REGION Network 7: FIXTURES NO DEFINE POSITION
   RUNG wire#powerrail
      Contact( "M_ONE" )
      wire#w1
      I_Contact( "DB4000_FIX_TABLE_POSITIONS".UNIT_01.FIXTURE_1.IN_LOAD_UNLOAD_STATION_1 )
      I_Contact( "DB4000_FIX_TABLE_POSITIONS".UNIT_01.FIXTURE_1.IN_SPARE_STATION_2 )
      I_Contact( "DB4000_FIX_TABLE_POSITIONS".UNIT_01.FIXTURE_1.IN_CLADDING_STATION_3 )
      I_Contact( "DB4000_FIX_TABLE_POSITIONS".UNIT_01.FIXTURE_1.IN_CLEAN_STATION_4 )
      Coil( "DB4000_FIX_TABLE_POSITIONS".UNIT_01.FIXTURE_1.NO_DEFINED_POSITION )
   END_RUNG
   RUNG wire#w1
      I_Contact( "DB4000_FIX_TABLE_POSITIONS".UNIT_01.FIXTURE_2.IN_LOAD_UNLOAD_STATION_1 )
      I_Contact( "DB4000_FIX_TABLE_POSITIONS".UNIT_01.FIXTURE_2.IN_SPARE_STATION_2 )
      I_Contact( "DB4000_FIX_TABLE_POSITIONS".UNIT_01.FIXTURE_2.IN_CLADDING_STATION_3 )
      I_Contact( "DB4000_FIX_TABLE_POSITIONS".UNIT_01.FIXTURE_2.IN_CLEAN_STATION_4 )
      Coil( "DB4000_FIX_TABLE_POSITIONS".UNIT_01.FIXTURE_2.NO_DEFINED_POSITION )
   END_RUNG
   RUNG wire#w1
      I_Contact( "DB4000_FIX_TABLE_POSITIONS".UNIT_01.FIXTURE_3.IN_LOAD_UNLOAD_STATION_1 )
      I_Contact( "DB4000_FIX_TABLE_POSITIONS".UNIT_01.FIXTURE_3.IN_SPARE_STATION_2 )
      I_Contact( "DB4000_FIX_TABLE_POSITIONS".UNIT_01.FIXTURE_3.IN_CLADDING_STATION_3 )
      I_Contact( "DB4000_FIX_TABLE_POSITIONS".UNIT_01.FIXTURE_3.IN_CLEAN_STATION_4 )
      Coil( "DB4000_FIX_TABLE_POSITIONS".UNIT_01.FIXTURE_3.NO_DEFINED_POSITION )
   END_RUNG
   RUNG wire#w1
      I_Contact( "DB4000_FIX_TABLE_POSITIONS".UNIT_01.FIXTURE_4.IN_LOAD_UNLOAD_STATION_1 )
      I_Contact( "DB4000_FIX_TABLE_POSITIONS".UNIT_01.FIXTURE_4.IN_SPARE_STATION_2 )
      I_Contact( "DB4000_FIX_TABLE_POSITIONS".UNIT_01.FIXTURE_4.IN_CLADDING_STATION_3 )
      I_Contact( "DB4000_FIX_TABLE_POSITIONS".UNIT_01.FIXTURE_4.IN_CLEAN_STATION_4 )
      Coil( "DB4000_FIX_TABLE_POSITIONS".UNIT_01.FIXTURE_4.NO_DEFINED_POSITION )
   END_RUNG
   // the same network as SCL:
   "DB4000_FIX_TABLE_POSITIONS".UNIT_01.FIXTURE_1.NO_DEFINED_POSITION := "M_ONE" AND NOT "DB4000_FIX_TABLE_POSITIONS".UNIT_01.FIXTURE_1.IN_LOAD_UNLOAD_STATION_1 AND NOT "DB4000_FIX_TABLE_POSITIONS".UNIT_01.FIXTURE_1.IN_SPARE_STATION_2 AND NOT "DB4000_FIX_TABLE_POSITIONS".UNIT_01.FIXTURE_1.IN_CLADDING_STATION_3 AND NOT "DB4000_FIX_TABLE_POSITIONS".UNIT_01.FIXTURE_1.IN_CLEAN_STATION_4;
   "DB4000_FIX_TABLE_POSITIONS".UNIT_01.FIXTURE_2.NO_DEFINED_POSITION := "M_ONE" AND NOT "DB4000_FIX_TABLE_POSITIONS".UNIT_01.FIXTURE_2.IN_LOAD_UNLOAD_STATION_1 AND NOT "DB4000_FIX_TABLE_POSITIONS".UNIT_01.FIXTURE_2.IN_SPARE_STATION_2 AND NOT "DB4000_FIX_TABLE_POSITIONS".UNIT_01.FIXTURE_2.IN_CLADDING_STATION_3 AND NOT "DB4000_FIX_TABLE_POSITIONS".UNIT_01.FIXTURE_2.IN_CLEAN_STATION_4;
   "DB4000_FIX_TABLE_POSITIONS".UNIT_01.FIXTURE_3.NO_DEFINED_POSITION := "M_ONE" AND NOT "DB4000_FIX_TABLE_POSITIONS".UNIT_01.FIXTURE_3.IN_LOAD_UNLOAD_STATION_1 AND NOT "DB4000_FIX_TABLE_POSITIONS".UNIT_01.FIXTURE_3.IN_SPARE_STATION_2 AND NOT "DB4000_FIX_TABLE_POSITIONS".UNIT_01.FIXTURE_3.IN_CLADDING_STATION_3 AND NOT "DB4000_FIX_TABLE_POSITIONS".UNIT_01.FIXTURE_3.IN_CLEAN_STATION_4;
   "DB4000_FIX_TABLE_POSITIONS".UNIT_01.FIXTURE_4.NO_DEFINED_POSITION := "M_ONE" AND NOT "DB4000_FIX_TABLE_POSITIONS".UNIT_01.FIXTURE_4.IN_LOAD_UNLOAD_STATION_1 AND NOT "DB4000_FIX_TABLE_POSITIONS".UNIT_01.FIXTURE_4.IN_SPARE_STATION_2 AND NOT "DB4000_FIX_TABLE_POSITIONS".UNIT_01.FIXTURE_4.IN_CLADDING_STATION_3 AND NOT "DB4000_FIX_TABLE_POSITIONS".UNIT_01.FIXTURE_4.IN_CLEAN_STATION_4;
END_REGION

REGION Network 8: AXIS E10 HOME POSITION
   RUNG wire#powerrail
      I_Contact( "DB131_CLADDING_AXIS_E10".SAFETY_POSITIONS.AX_POS_0_DEGREES.IN_POSITION )
      I_Contact( "DB131_CLADDING_AXIS_E10".SAFETY_POSITIONS.AX_POS_90_DEGREES.IN_POSITION )
      I_Contact( "DB131_CLADDING_AXIS_E10".SAFETY_POSITIONS.AX_POS_180_DEGREES.IN_POSITION )
      I_Contact( "DB131_CLADDING_AXIS_E10".SAFETY_POSITIONS.AX_POS_270_DEGREES.IN_POSITION )
      Not()
      Coil( "DB4000_FIX_TABLE_POSITIONS".UNIT_01.AXIS_E10_HOME_POS )
   END_RUNG
   // the same network as SCL:
   "DB4000_FIX_TABLE_POSITIONS".UNIT_01.AXIS_E10_HOME_POS := NOT (NOT "DB131_CLADDING_AXIS_E10".SAFETY_POSITIONS.AX_POS_0_DEGREES.IN_POSITION AND NOT "DB131_CLADDING_AXIS_E10".SAFETY_POSITIONS.AX_POS_90_DEGREES.IN_POSITION AND NOT "DB131_CLADDING_AXIS_E10".SAFETY_POSITIONS.AX_POS_180_DEGREES.IN_POSITION AND NOT "DB131_CLADDING_AXIS_E10".SAFETY_POSITIONS.AX_POS_270_DEGREES.IN_POSITION);
END_REGION

REGION Network 9: AXIS E10 NOT IN A DEFINED POSITION
   RUNG wire#powerrail
      I_Contact( "DB131_CLADDING_AXIS_E10".SAFETY_POSITIONS.AX_POS_0_DEGREES.IN_POSITION )
      I_Contact( "DB131_CLADDING_AXIS_E10".SAFETY_POSITIONS.AX_POS_90_DEGREES.IN_POSITION )
      I_Contact( "DB131_CLADDING_AXIS_E10".SAFETY_POSITIONS.AX_POS_180_DEGREES.IN_POSITION )
      I_Contact( "DB131_CLADDING_AXIS_E10".SAFETY_POSITIONS.AX_POS_270_DEGREES.IN_POSITION )
      Coil( "DB4000_FIX_TABLE_POSITIONS".UNIT_01.AXIS_E10_NOT_DEFINED_POS )
   END_RUNG
   // the same network as SCL:
   "DB4000_FIX_TABLE_POSITIONS".UNIT_01.AXIS_E10_NOT_DEFINED_POS := NOT "DB131_CLADDING_AXIS_E10".SAFETY_POSITIONS.AX_POS_0_DEGREES.IN_POSITION AND NOT "DB131_CLADDING_AXIS_E10".SAFETY_POSITIONS.AX_POS_90_DEGREES.IN_POSITION AND NOT "DB131_CLADDING_AXIS_E10".SAFETY_POSITIONS.AX_POS_180_DEGREES.IN_POSITION AND NOT "DB131_CLADDING_AXIS_E10".SAFETY_POSITIONS.AX_POS_270_DEGREES.IN_POSITION;
END_REGION

REGION Network 10: <<<<<<<<<<<<<<<<<<<< UNIT 02 >>>>>>>>>>>>>>>>>>>>
END_REGION

REGION Network 11: AXIS E20 0 DEGREES
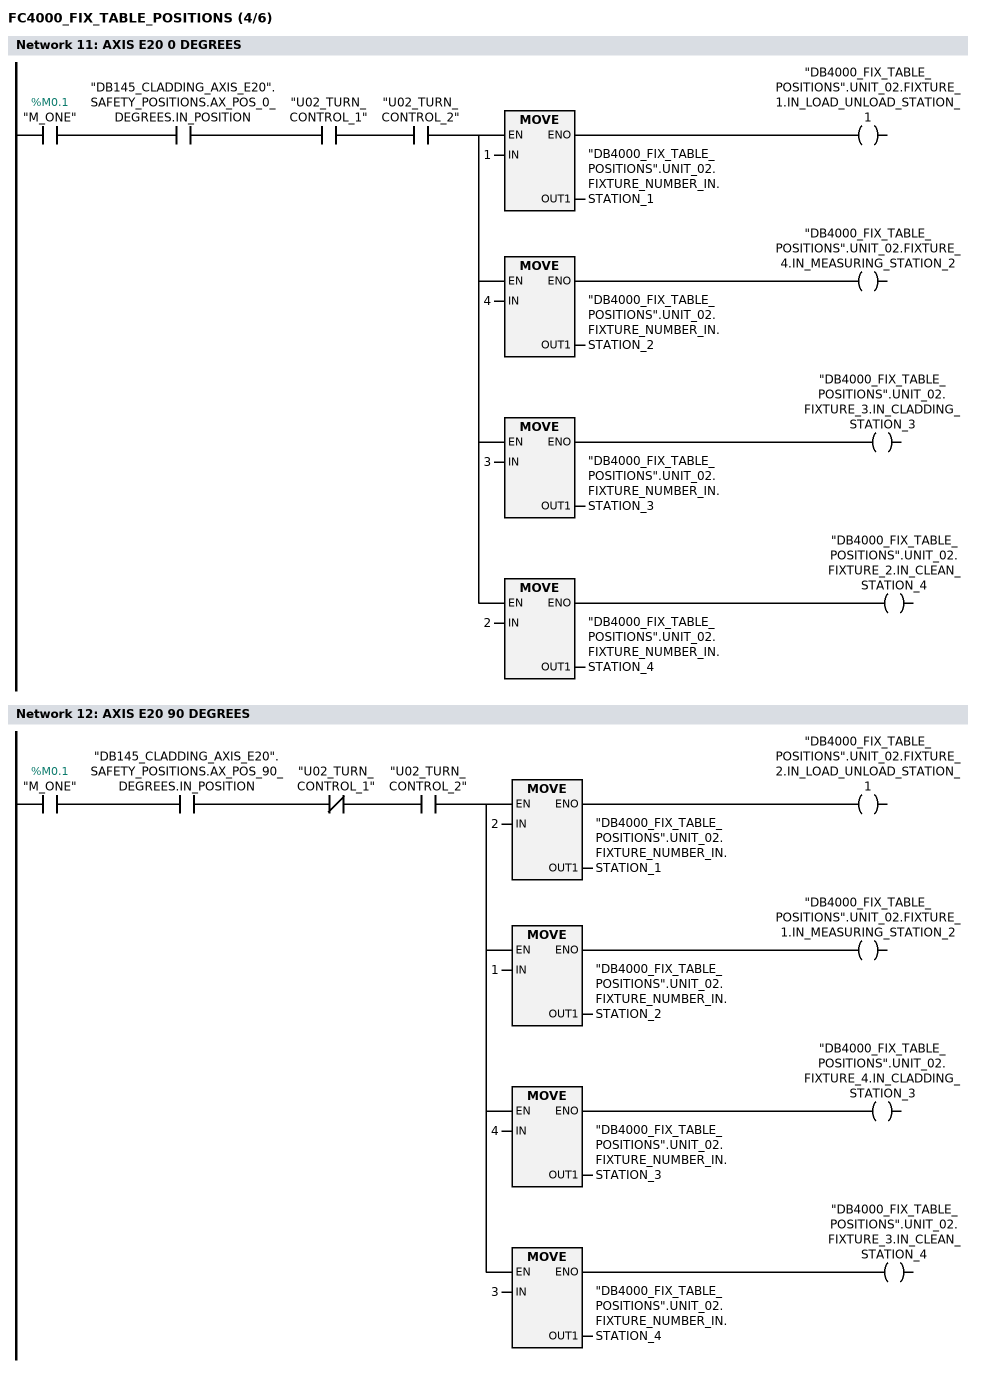
   RUNG wire#powerrail
      Contact( "M_ONE" )
      Contact( "DB145_CLADDING_AXIS_E20".SAFETY_POSITIONS.AX_POS_0_DEGREES.IN_POSITION )
      Contact( "U02_TURN_CONTROL_1" )
      Contact( "U02_TURN_CONTROL_2" )
      wire#w1
      Move(in := 1, out1 => "DB4000_FIX_TABLE_POSITIONS".UNIT_02.FIXTURE_NUMBER_IN.STATION_1)
      Coil( "DB4000_FIX_TABLE_POSITIONS".UNIT_02.FIXTURE_1.IN_LOAD_UNLOAD_STATION_1 )
   END_RUNG
   RUNG wire#w1
      Move(in := 4, out1 => "DB4000_FIX_TABLE_POSITIONS".UNIT_02.FIXTURE_NUMBER_IN.STATION_2)
      Coil( "DB4000_FIX_TABLE_POSITIONS".UNIT_02.FIXTURE_4.IN_MEASURING_STATION_2 )
   END_RUNG
   RUNG wire#w1
      Move(in := 3, out1 => "DB4000_FIX_TABLE_POSITIONS".UNIT_02.FIXTURE_NUMBER_IN.STATION_3)
      Coil( "DB4000_FIX_TABLE_POSITIONS".UNIT_02.FIXTURE_3.IN_CLADDING_STATION_3 )
   END_RUNG
   RUNG wire#w1
      Move(in := 2, out1 => "DB4000_FIX_TABLE_POSITIONS".UNIT_02.FIXTURE_NUMBER_IN.STATION_4)
      Coil( "DB4000_FIX_TABLE_POSITIONS".UNIT_02.FIXTURE_2.IN_CLEAN_STATION_4 )
   END_RUNG
   // the same network as SCL:
   #_w1 := "M_ONE" AND "DB145_CLADDING_AXIS_E20".SAFETY_POSITIONS.AX_POS_0_DEGREES.IN_POSITION AND "U02_TURN_CONTROL_1" AND "U02_TURN_CONTROL_2";
   IF #_w1 THEN "DB4000_FIX_TABLE_POSITIONS".UNIT_02.FIXTURE_NUMBER_IN.STATION_1 := 1; END_IF;
   "DB4000_FIX_TABLE_POSITIONS".UNIT_02.FIXTURE_1.IN_LOAD_UNLOAD_STATION_1 := #_w1;
   IF #_w1 THEN "DB4000_FIX_TABLE_POSITIONS".UNIT_02.FIXTURE_NUMBER_IN.STATION_2 := 4; END_IF;
   "DB4000_FIX_TABLE_POSITIONS".UNIT_02.FIXTURE_4.IN_MEASURING_STATION_2 := #_w1;
   IF #_w1 THEN "DB4000_FIX_TABLE_POSITIONS".UNIT_02.FIXTURE_NUMBER_IN.STATION_3 := 3; END_IF;
   "DB4000_FIX_TABLE_POSITIONS".UNIT_02.FIXTURE_3.IN_CLADDING_STATION_3 := #_w1;
   IF #_w1 THEN "DB4000_FIX_TABLE_POSITIONS".UNIT_02.FIXTURE_NUMBER_IN.STATION_4 := 2; END_IF;
   "DB4000_FIX_TABLE_POSITIONS".UNIT_02.FIXTURE_2.IN_CLEAN_STATION_4 := #_w1;
END_REGION

REGION Network 12: AXIS E20 90 DEGREES
   RUNG wire#powerrail
      Contact( "M_ONE" )
      Contact( "DB145_CLADDING_AXIS_E20".SAFETY_POSITIONS.AX_POS_90_DEGREES.IN_POSITION )
      I_Contact( "U02_TURN_CONTROL_1" )
      Contact( "U02_TURN_CONTROL_2" )
      wire#w1
      Move(in := 2, out1 => "DB4000_FIX_TABLE_POSITIONS".UNIT_02.FIXTURE_NUMBER_IN.STATION_1)
      Coil( "DB4000_FIX_TABLE_POSITIONS".UNIT_02.FIXTURE_2.IN_LOAD_UNLOAD_STATION_1 )
   END_RUNG
   RUNG wire#w1
      Move(in := 1, out1 => "DB4000_FIX_TABLE_POSITIONS".UNIT_02.FIXTURE_NUMBER_IN.STATION_2)
      Coil( "DB4000_FIX_TABLE_POSITIONS".UNIT_02.FIXTURE_1.IN_MEASURING_STATION_2 )
   END_RUNG
   RUNG wire#w1
      Move(in := 4, out1 => "DB4000_FIX_TABLE_POSITIONS".UNIT_02.FIXTURE_NUMBER_IN.STATION_3)
      Coil( "DB4000_FIX_TABLE_POSITIONS".UNIT_02.FIXTURE_4.IN_CLADDING_STATION_3 )
   END_RUNG
   RUNG wire#w1
      Move(in := 3, out1 => "DB4000_FIX_TABLE_POSITIONS".UNIT_02.FIXTURE_NUMBER_IN.STATION_4)
      Coil( "DB4000_FIX_TABLE_POSITIONS".UNIT_02.FIXTURE_3.IN_CLEAN_STATION_4 )
   END_RUNG
   // the same network as SCL:
   #_w1 := "M_ONE" AND "DB145_CLADDING_AXIS_E20".SAFETY_POSITIONS.AX_POS_90_DEGREES.IN_POSITION AND NOT "U02_TURN_CONTROL_1" AND "U02_TURN_CONTROL_2";
   IF #_w1 THEN "DB4000_FIX_TABLE_POSITIONS".UNIT_02.FIXTURE_NUMBER_IN.STATION_1 := 2; END_IF;
   "DB4000_FIX_TABLE_POSITIONS".UNIT_02.FIXTURE_2.IN_LOAD_UNLOAD_STATION_1 := #_w1;
   IF #_w1 THEN "DB4000_FIX_TABLE_POSITIONS".UNIT_02.FIXTURE_NUMBER_IN.STATION_2 := 1; END_IF;
   "DB4000_FIX_TABLE_POSITIONS".UNIT_02.FIXTURE_1.IN_MEASURING_STATION_2 := #_w1;
   IF #_w1 THEN "DB4000_FIX_TABLE_POSITIONS".UNIT_02.FIXTURE_NUMBER_IN.STATION_3 := 4; END_IF;
   "DB4000_FIX_TABLE_POSITIONS".UNIT_02.FIXTURE_4.IN_CLADDING_STATION_3 := #_w1;
   IF #_w1 THEN "DB4000_FIX_TABLE_POSITIONS".UNIT_02.FIXTURE_NUMBER_IN.STATION_4 := 3; END_IF;
   "DB4000_FIX_TABLE_POSITIONS".UNIT_02.FIXTURE_3.IN_CLEAN_STATION_4 := #_w1;
END_REGION

REGION Network 13: AXIS E20 180 DEGREES
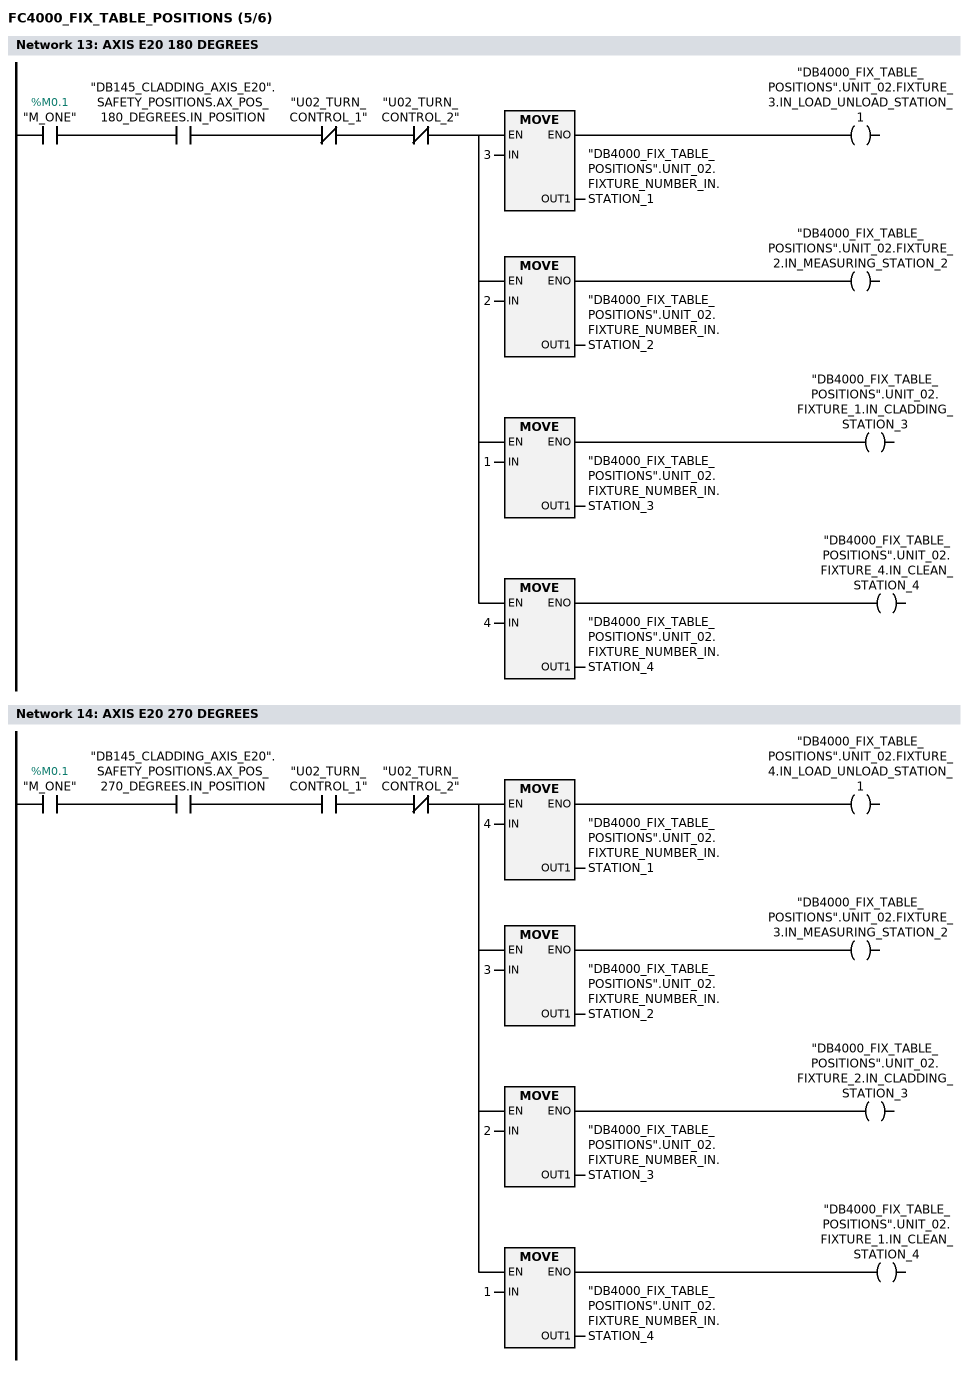
   RUNG wire#powerrail
      Contact( "M_ONE" )
      Contact( "DB145_CLADDING_AXIS_E20".SAFETY_POSITIONS.AX_POS_180_DEGREES.IN_POSITION )
      I_Contact( "U02_TURN_CONTROL_1" )
      I_Contact( "U02_TURN_CONTROL_2" )
      wire#w1
      Move(in := 3, out1 => "DB4000_FIX_TABLE_POSITIONS".UNIT_02.FIXTURE_NUMBER_IN.STATION_1)
      Coil( "DB4000_FIX_TABLE_POSITIONS".UNIT_02.FIXTURE_3.IN_LOAD_UNLOAD_STATION_1 )
   END_RUNG
   RUNG wire#w1
      Move(in := 2, out1 => "DB4000_FIX_TABLE_POSITIONS".UNIT_02.FIXTURE_NUMBER_IN.STATION_2)
      Coil( "DB4000_FIX_TABLE_POSITIONS".UNIT_02.FIXTURE_2.IN_MEASURING_STATION_2 )
   END_RUNG
   RUNG wire#w1
      Move(in := 1, out1 => "DB4000_FIX_TABLE_POSITIONS".UNIT_02.FIXTURE_NUMBER_IN.STATION_3)
      Coil( "DB4000_FIX_TABLE_POSITIONS".UNIT_02.FIXTURE_1.IN_CLADDING_STATION_3 )
   END_RUNG
   RUNG wire#w1
      Move(in := 4, out1 => "DB4000_FIX_TABLE_POSITIONS".UNIT_02.FIXTURE_NUMBER_IN.STATION_4)
      Coil( "DB4000_FIX_TABLE_POSITIONS".UNIT_02.FIXTURE_4.IN_CLEAN_STATION_4 )
   END_RUNG
   // the same network as SCL:
   #_w1 := "M_ONE" AND "DB145_CLADDING_AXIS_E20".SAFETY_POSITIONS.AX_POS_180_DEGREES.IN_POSITION AND NOT "U02_TURN_CONTROL_1" AND NOT "U02_TURN_CONTROL_2";
   IF #_w1 THEN "DB4000_FIX_TABLE_POSITIONS".UNIT_02.FIXTURE_NUMBER_IN.STATION_1 := 3; END_IF;
   "DB4000_FIX_TABLE_POSITIONS".UNIT_02.FIXTURE_3.IN_LOAD_UNLOAD_STATION_1 := #_w1;
   IF #_w1 THEN "DB4000_FIX_TABLE_POSITIONS".UNIT_02.FIXTURE_NUMBER_IN.STATION_2 := 2; END_IF;
   "DB4000_FIX_TABLE_POSITIONS".UNIT_02.FIXTURE_2.IN_MEASURING_STATION_2 := #_w1;
   IF #_w1 THEN "DB4000_FIX_TABLE_POSITIONS".UNIT_02.FIXTURE_NUMBER_IN.STATION_3 := 1; END_IF;
   "DB4000_FIX_TABLE_POSITIONS".UNIT_02.FIXTURE_1.IN_CLADDING_STATION_3 := #_w1;
   IF #_w1 THEN "DB4000_FIX_TABLE_POSITIONS".UNIT_02.FIXTURE_NUMBER_IN.STATION_4 := 4; END_IF;
   "DB4000_FIX_TABLE_POSITIONS".UNIT_02.FIXTURE_4.IN_CLEAN_STATION_4 := #_w1;
END_REGION

REGION Network 14: AXIS E20 270 DEGREES
   RUNG wire#powerrail
      Contact( "M_ONE" )
      Contact( "DB145_CLADDING_AXIS_E20".SAFETY_POSITIONS.AX_POS_270_DEGREES.IN_POSITION )
      Contact( "U02_TURN_CONTROL_1" )
      I_Contact( "U02_TURN_CONTROL_2" )
      wire#w1
      Move(in := 4, out1 => "DB4000_FIX_TABLE_POSITIONS".UNIT_02.FIXTURE_NUMBER_IN.STATION_1)
      Coil( "DB4000_FIX_TABLE_POSITIONS".UNIT_02.FIXTURE_4.IN_LOAD_UNLOAD_STATION_1 )
   END_RUNG
   RUNG wire#w1
      Move(in := 3, out1 => "DB4000_FIX_TABLE_POSITIONS".UNIT_02.FIXTURE_NUMBER_IN.STATION_2)
      Coil( "DB4000_FIX_TABLE_POSITIONS".UNIT_02.FIXTURE_3.IN_MEASURING_STATION_2 )
   END_RUNG
   RUNG wire#w1
      Move(in := 2, out1 => "DB4000_FIX_TABLE_POSITIONS".UNIT_02.FIXTURE_NUMBER_IN.STATION_3)
      Coil( "DB4000_FIX_TABLE_POSITIONS".UNIT_02.FIXTURE_2.IN_CLADDING_STATION_3 )
   END_RUNG
   RUNG wire#w1
      Move(in := 1, out1 => "DB4000_FIX_TABLE_POSITIONS".UNIT_02.FIXTURE_NUMBER_IN.STATION_4)
      Coil( "DB4000_FIX_TABLE_POSITIONS".UNIT_02.FIXTURE_1.IN_CLEAN_STATION_4 )
   END_RUNG
   // the same network as SCL:
   #_w1 := "M_ONE" AND "DB145_CLADDING_AXIS_E20".SAFETY_POSITIONS.AX_POS_270_DEGREES.IN_POSITION AND "U02_TURN_CONTROL_1" AND NOT "U02_TURN_CONTROL_2";
   IF #_w1 THEN "DB4000_FIX_TABLE_POSITIONS".UNIT_02.FIXTURE_NUMBER_IN.STATION_1 := 4; END_IF;
   "DB4000_FIX_TABLE_POSITIONS".UNIT_02.FIXTURE_4.IN_LOAD_UNLOAD_STATION_1 := #_w1;
   IF #_w1 THEN "DB4000_FIX_TABLE_POSITIONS".UNIT_02.FIXTURE_NUMBER_IN.STATION_2 := 3; END_IF;
   "DB4000_FIX_TABLE_POSITIONS".UNIT_02.FIXTURE_3.IN_MEASURING_STATION_2 := #_w1;
   IF #_w1 THEN "DB4000_FIX_TABLE_POSITIONS".UNIT_02.FIXTURE_NUMBER_IN.STATION_3 := 2; END_IF;
   "DB4000_FIX_TABLE_POSITIONS".UNIT_02.FIXTURE_2.IN_CLADDING_STATION_3 := #_w1;
   IF #_w1 THEN "DB4000_FIX_TABLE_POSITIONS".UNIT_02.FIXTURE_NUMBER_IN.STATION_4 := 1; END_IF;
   "DB4000_FIX_TABLE_POSITIONS".UNIT_02.FIXTURE_1.IN_CLEAN_STATION_4 := #_w1;
END_REGION

REGION Network 15: E20 AXIS POSITION REACH
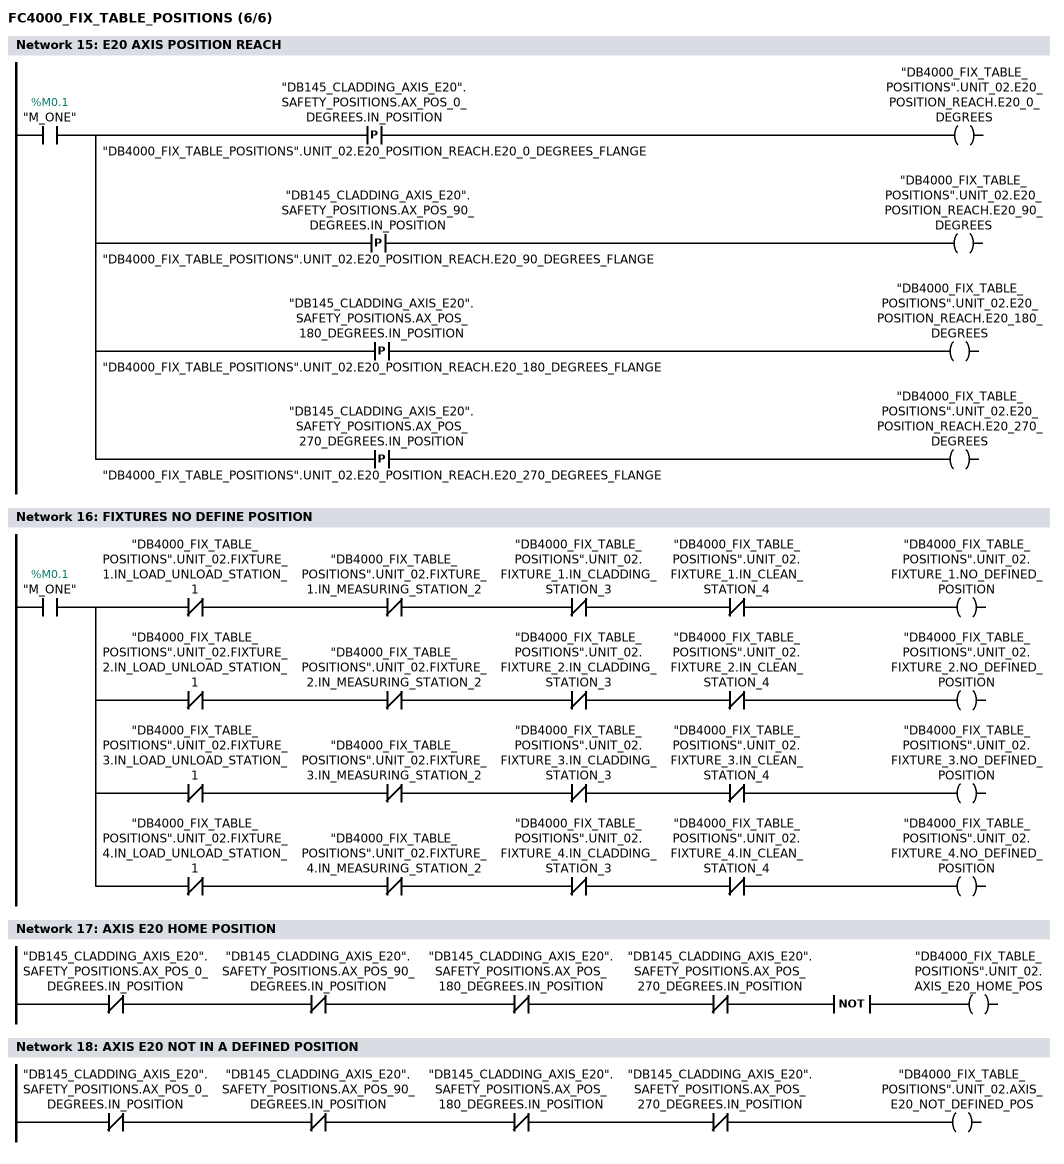
   RUNG wire#powerrail
      Contact( "M_ONE" )
      wire#w1
      P_Contact(operand := "DB145_CLADDING_AXIS_E20".SAFETY_POSITIONS.AX_POS_0_DEGREES.IN_POSITION, bit := "DB4000_FIX_TABLE_POSITIONS".UNIT_02.E20_POSITION_REACH.E20_0_DEGREES_FLANGE)
      Coil( "DB4000_FIX_TABLE_POSITIONS".UNIT_02.E20_POSITION_REACH.E20_0_DEGREES )
   END_RUNG
   RUNG wire#w1
      P_Contact(operand := "DB145_CLADDING_AXIS_E20".SAFETY_POSITIONS.AX_POS_90_DEGREES.IN_POSITION, bit := "DB4000_FIX_TABLE_POSITIONS".UNIT_02.E20_POSITION_REACH.E20_90_DEGREES_FLANGE)
      Coil( "DB4000_FIX_TABLE_POSITIONS".UNIT_02.E20_POSITION_REACH.E20_90_DEGREES )
   END_RUNG
   RUNG wire#w1
      P_Contact(operand := "DB145_CLADDING_AXIS_E20".SAFETY_POSITIONS.AX_POS_180_DEGREES.IN_POSITION, bit := "DB4000_FIX_TABLE_POSITIONS".UNIT_02.E20_POSITION_REACH.E20_180_DEGREES_FLANGE)
      Coil( "DB4000_FIX_TABLE_POSITIONS".UNIT_02.E20_POSITION_REACH.E20_180_DEGREES )
   END_RUNG
   RUNG wire#w1
      P_Contact(operand := "DB145_CLADDING_AXIS_E20".SAFETY_POSITIONS.AX_POS_270_DEGREES.IN_POSITION, bit := "DB4000_FIX_TABLE_POSITIONS".UNIT_02.E20_POSITION_REACH.E20_270_DEGREES_FLANGE)
      Coil( "DB4000_FIX_TABLE_POSITIONS".UNIT_02.E20_POSITION_REACH.E20_270_DEGREES )
   END_RUNG
   // the same network as SCL:
   #_w1 := "M_ONE" AND "DB145_CLADDING_AXIS_E20".SAFETY_POSITIONS.AX_POS_0_DEGREES.IN_POSITION AND NOT "DB4000_FIX_TABLE_POSITIONS".UNIT_02.E20_POSITION_REACH.E20_0_DEGREES_FLANGE;   // rising edge of "DB145_CLADDING_AXIS_E20".SAFETY_POSITIONS.AX_POS_0_DEGREES.IN_POSITION
   "DB4000_FIX_TABLE_POSITIONS".UNIT_02.E20_POSITION_REACH.E20_0_DEGREES_FLANGE := "DB145_CLADDING_AXIS_E20".SAFETY_POSITIONS.AX_POS_0_DEGREES.IN_POSITION;
   "DB4000_FIX_TABLE_POSITIONS".UNIT_02.E20_POSITION_REACH.E20_0_DEGREES := #_w1;
   #_w2 := "M_ONE" AND "DB145_CLADDING_AXIS_E20".SAFETY_POSITIONS.AX_POS_90_DEGREES.IN_POSITION AND NOT "DB4000_FIX_TABLE_POSITIONS".UNIT_02.E20_POSITION_REACH.E20_90_DEGREES_FLANGE;   // rising edge of "DB145_CLADDING_AXIS_E20".SAFETY_POSITIONS.AX_POS_90_DEGREES.IN_POSITION
   "DB4000_FIX_TABLE_POSITIONS".UNIT_02.E20_POSITION_REACH.E20_90_DEGREES_FLANGE := "DB145_CLADDING_AXIS_E20".SAFETY_POSITIONS.AX_POS_90_DEGREES.IN_POSITION;
   "DB4000_FIX_TABLE_POSITIONS".UNIT_02.E20_POSITION_REACH.E20_90_DEGREES := #_w2;
   #_w3 := "M_ONE" AND "DB145_CLADDING_AXIS_E20".SAFETY_POSITIONS.AX_POS_180_DEGREES.IN_POSITION AND NOT "DB4000_FIX_TABLE_POSITIONS".UNIT_02.E20_POSITION_REACH.E20_180_DEGREES_FLANGE;   // rising edge of "DB145_CLADDING_AXIS_E20".SAFETY_POSITIONS.AX_POS_180_DEGREES.IN_POSITION
   "DB4000_FIX_TABLE_POSITIONS".UNIT_02.E20_POSITION_REACH.E20_180_DEGREES_FLANGE := "DB145_CLADDING_AXIS_E20".SAFETY_POSITIONS.AX_POS_180_DEGREES.IN_POSITION;
   "DB4000_FIX_TABLE_POSITIONS".UNIT_02.E20_POSITION_REACH.E20_180_DEGREES := #_w3;
   #_w4 := "M_ONE" AND "DB145_CLADDING_AXIS_E20".SAFETY_POSITIONS.AX_POS_270_DEGREES.IN_POSITION AND NOT "DB4000_FIX_TABLE_POSITIONS".UNIT_02.E20_POSITION_REACH.E20_270_DEGREES_FLANGE;   // rising edge of "DB145_CLADDING_AXIS_E20".SAFETY_POSITIONS.AX_POS_270_DEGREES.IN_POSITION
   "DB4000_FIX_TABLE_POSITIONS".UNIT_02.E20_POSITION_REACH.E20_270_DEGREES_FLANGE := "DB145_CLADDING_AXIS_E20".SAFETY_POSITIONS.AX_POS_270_DEGREES.IN_POSITION;
   "DB4000_FIX_TABLE_POSITIONS".UNIT_02.E20_POSITION_REACH.E20_270_DEGREES := #_w4;
END_REGION

REGION Network 16: FIXTURES NO DEFINE POSITION
   RUNG wire#powerrail
      Contact( "M_ONE" )
      wire#w1
      I_Contact( "DB4000_FIX_TABLE_POSITIONS".UNIT_02.FIXTURE_1.IN_LOAD_UNLOAD_STATION_1 )
      I_Contact( "DB4000_FIX_TABLE_POSITIONS".UNIT_02.FIXTURE_1.IN_MEASURING_STATION_2 )
      I_Contact( "DB4000_FIX_TABLE_POSITIONS".UNIT_02.FIXTURE_1.IN_CLADDING_STATION_3 )
      I_Contact( "DB4000_FIX_TABLE_POSITIONS".UNIT_02.FIXTURE_1.IN_CLEAN_STATION_4 )
      Coil( "DB4000_FIX_TABLE_POSITIONS".UNIT_02.FIXTURE_1.NO_DEFINED_POSITION )
   END_RUNG
   RUNG wire#w1
      I_Contact( "DB4000_FIX_TABLE_POSITIONS".UNIT_02.FIXTURE_2.IN_LOAD_UNLOAD_STATION_1 )
      I_Contact( "DB4000_FIX_TABLE_POSITIONS".UNIT_02.FIXTURE_2.IN_MEASURING_STATION_2 )
      I_Contact( "DB4000_FIX_TABLE_POSITIONS".UNIT_02.FIXTURE_2.IN_CLADDING_STATION_3 )
      I_Contact( "DB4000_FIX_TABLE_POSITIONS".UNIT_02.FIXTURE_2.IN_CLEAN_STATION_4 )
      Coil( "DB4000_FIX_TABLE_POSITIONS".UNIT_02.FIXTURE_2.NO_DEFINED_POSITION )
   END_RUNG
   RUNG wire#w1
      I_Contact( "DB4000_FIX_TABLE_POSITIONS".UNIT_02.FIXTURE_3.IN_LOAD_UNLOAD_STATION_1 )
      I_Contact( "DB4000_FIX_TABLE_POSITIONS".UNIT_02.FIXTURE_3.IN_MEASURING_STATION_2 )
      I_Contact( "DB4000_FIX_TABLE_POSITIONS".UNIT_02.FIXTURE_3.IN_CLADDING_STATION_3 )
      I_Contact( "DB4000_FIX_TABLE_POSITIONS".UNIT_02.FIXTURE_3.IN_CLEAN_STATION_4 )
      Coil( "DB4000_FIX_TABLE_POSITIONS".UNIT_02.FIXTURE_3.NO_DEFINED_POSITION )
   END_RUNG
   RUNG wire#w1
      I_Contact( "DB4000_FIX_TABLE_POSITIONS".UNIT_02.FIXTURE_4.IN_LOAD_UNLOAD_STATION_1 )
      I_Contact( "DB4000_FIX_TABLE_POSITIONS".UNIT_02.FIXTURE_4.IN_MEASURING_STATION_2 )
      I_Contact( "DB4000_FIX_TABLE_POSITIONS".UNIT_02.FIXTURE_4.IN_CLADDING_STATION_3 )
      I_Contact( "DB4000_FIX_TABLE_POSITIONS".UNIT_02.FIXTURE_4.IN_CLEAN_STATION_4 )
      Coil( "DB4000_FIX_TABLE_POSITIONS".UNIT_02.FIXTURE_4.NO_DEFINED_POSITION )
   END_RUNG
   // the same network as SCL:
   "DB4000_FIX_TABLE_POSITIONS".UNIT_02.FIXTURE_1.NO_DEFINED_POSITION := "M_ONE" AND NOT "DB4000_FIX_TABLE_POSITIONS".UNIT_02.FIXTURE_1.IN_LOAD_UNLOAD_STATION_1 AND NOT "DB4000_FIX_TABLE_POSITIONS".UNIT_02.FIXTURE_1.IN_MEASURING_STATION_2 AND NOT "DB4000_FIX_TABLE_POSITIONS".UNIT_02.FIXTURE_1.IN_CLADDING_STATION_3 AND NOT "DB4000_FIX_TABLE_POSITIONS".UNIT_02.FIXTURE_1.IN_CLEAN_STATION_4;
   "DB4000_FIX_TABLE_POSITIONS".UNIT_02.FIXTURE_2.NO_DEFINED_POSITION := "M_ONE" AND NOT "DB4000_FIX_TABLE_POSITIONS".UNIT_02.FIXTURE_2.IN_LOAD_UNLOAD_STATION_1 AND NOT "DB4000_FIX_TABLE_POSITIONS".UNIT_02.FIXTURE_2.IN_MEASURING_STATION_2 AND NOT "DB4000_FIX_TABLE_POSITIONS".UNIT_02.FIXTURE_2.IN_CLADDING_STATION_3 AND NOT "DB4000_FIX_TABLE_POSITIONS".UNIT_02.FIXTURE_2.IN_CLEAN_STATION_4;
   "DB4000_FIX_TABLE_POSITIONS".UNIT_02.FIXTURE_3.NO_DEFINED_POSITION := "M_ONE" AND NOT "DB4000_FIX_TABLE_POSITIONS".UNIT_02.FIXTURE_3.IN_LOAD_UNLOAD_STATION_1 AND NOT "DB4000_FIX_TABLE_POSITIONS".UNIT_02.FIXTURE_3.IN_MEASURING_STATION_2 AND NOT "DB4000_FIX_TABLE_POSITIONS".UNIT_02.FIXTURE_3.IN_CLADDING_STATION_3 AND NOT "DB4000_FIX_TABLE_POSITIONS".UNIT_02.FIXTURE_3.IN_CLEAN_STATION_4;
   "DB4000_FIX_TABLE_POSITIONS".UNIT_02.FIXTURE_4.NO_DEFINED_POSITION := "M_ONE" AND NOT "DB4000_FIX_TABLE_POSITIONS".UNIT_02.FIXTURE_4.IN_LOAD_UNLOAD_STATION_1 AND NOT "DB4000_FIX_TABLE_POSITIONS".UNIT_02.FIXTURE_4.IN_MEASURING_STATION_2 AND NOT "DB4000_FIX_TABLE_POSITIONS".UNIT_02.FIXTURE_4.IN_CLADDING_STATION_3 AND NOT "DB4000_FIX_TABLE_POSITIONS".UNIT_02.FIXTURE_4.IN_CLEAN_STATION_4;
END_REGION

REGION Network 17: AXIS E20 HOME POSITION
   RUNG wire#powerrail
      I_Contact( "DB145_CLADDING_AXIS_E20".SAFETY_POSITIONS.AX_POS_0_DEGREES.IN_POSITION )
      I_Contact( "DB145_CLADDING_AXIS_E20".SAFETY_POSITIONS.AX_POS_90_DEGREES.IN_POSITION )
      I_Contact( "DB145_CLADDING_AXIS_E20".SAFETY_POSITIONS.AX_POS_180_DEGREES.IN_POSITION )
      I_Contact( "DB145_CLADDING_AXIS_E20".SAFETY_POSITIONS.AX_POS_270_DEGREES.IN_POSITION )
      Not()
      Coil( "DB4000_FIX_TABLE_POSITIONS".UNIT_02.AXIS_E20_HOME_POS )
   END_RUNG
   // the same network as SCL:
   "DB4000_FIX_TABLE_POSITIONS".UNIT_02.AXIS_E20_HOME_POS := NOT (NOT "DB145_CLADDING_AXIS_E20".SAFETY_POSITIONS.AX_POS_0_DEGREES.IN_POSITION AND NOT "DB145_CLADDING_AXIS_E20".SAFETY_POSITIONS.AX_POS_90_DEGREES.IN_POSITION AND NOT "DB145_CLADDING_AXIS_E20".SAFETY_POSITIONS.AX_POS_180_DEGREES.IN_POSITION AND NOT "DB145_CLADDING_AXIS_E20".SAFETY_POSITIONS.AX_POS_270_DEGREES.IN_POSITION);
END_REGION

REGION Network 18: AXIS E20 NOT IN A DEFINED POSITION
   RUNG wire#powerrail
      I_Contact( "DB145_CLADDING_AXIS_E20".SAFETY_POSITIONS.AX_POS_0_DEGREES.IN_POSITION )
      I_Contact( "DB145_CLADDING_AXIS_E20".SAFETY_POSITIONS.AX_POS_90_DEGREES.IN_POSITION )
      I_Contact( "DB145_CLADDING_AXIS_E20".SAFETY_POSITIONS.AX_POS_180_DEGREES.IN_POSITION )
      I_Contact( "DB145_CLADDING_AXIS_E20".SAFETY_POSITIONS.AX_POS_270_DEGREES.IN_POSITION )
      Coil( "DB4000_FIX_TABLE_POSITIONS".UNIT_02.AXIS_E20_NOT_DEFINED_POS )
   END_RUNG
   // the same network as SCL:
   "DB4000_FIX_TABLE_POSITIONS".UNIT_02.AXIS_E20_NOT_DEFINED_POS := NOT "DB145_CLADDING_AXIS_E20".SAFETY_POSITIONS.AX_POS_0_DEGREES.IN_POSITION AND NOT "DB145_CLADDING_AXIS_E20".SAFETY_POSITIONS.AX_POS_90_DEGREES.IN_POSITION AND NOT "DB145_CLADDING_AXIS_E20".SAFETY_POSITIONS.AX_POS_180_DEGREES.IN_POSITION AND NOT "DB145_CLADDING_AXIS_E20".SAFETY_POSITIONS.AX_POS_270_DEGREES.IN_POSITION;
END_REGION
END_FUNCTION

FUNCTION "FC4001_FIXTURES_CALIBRATION" : Void   // FC4001, LAD
{ S7_Optimized_Access := 'TRUE' }
VERSION : 0.1
// stored: AutoNumber false, IsIECCheckEnabled false, SetENOAutomatically false, UDAEnableTagReadback false
BEGIN

REGION Network 1: FIXTURE 1 STATION 2 CALIBRATION DONE MEMORY
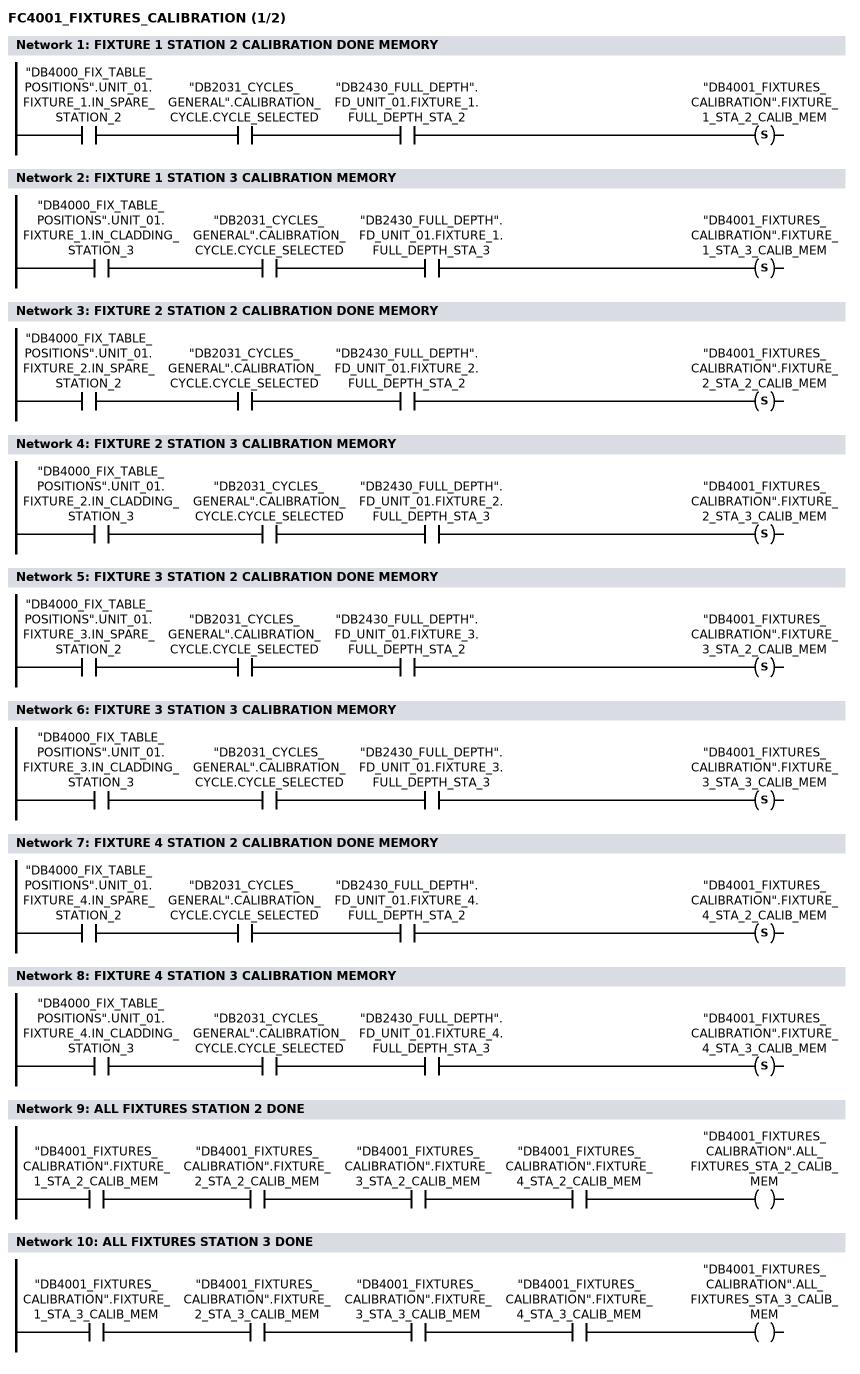
   RUNG wire#powerrail
      Contact( "DB4000_FIX_TABLE_POSITIONS".UNIT_01.FIXTURE_1.IN_SPARE_STATION_2 )
      Contact( "DB2031_CYCLES_GENERAL".CALIBRATION_CYCLE.CYCLE_SELECTED )
      Contact( "DB2430_FULL_DEPTH".FD_UNIT_01.FIXTURE_1.FULL_DEPTH_STA_2 )
      S_Coil( "DB4001_FIXTURES_CALIBRATION".FIXTURE_1_STA_2_CALIB_MEM )
   END_RUNG
   // the same network as SCL:
   IF "DB4000_FIX_TABLE_POSITIONS".UNIT_01.FIXTURE_1.IN_SPARE_STATION_2 AND "DB2031_CYCLES_GENERAL".CALIBRATION_CYCLE.CYCLE_SELECTED AND "DB2430_FULL_DEPTH".FD_UNIT_01.FIXTURE_1.FULL_DEPTH_STA_2 THEN
       "DB4001_FIXTURES_CALIBRATION".FIXTURE_1_STA_2_CALIB_MEM := TRUE;
   END_IF;
END_REGION

REGION Network 2: FIXTURE 1 STATION 3 CALIBRATION MEMORY
   RUNG wire#powerrail
      Contact( "DB4000_FIX_TABLE_POSITIONS".UNIT_01.FIXTURE_1.IN_CLADDING_STATION_3 )
      Contact( "DB2031_CYCLES_GENERAL".CALIBRATION_CYCLE.CYCLE_SELECTED )
      Contact( "DB2430_FULL_DEPTH".FD_UNIT_01.FIXTURE_1.FULL_DEPTH_STA_3 )
      S_Coil( "DB4001_FIXTURES_CALIBRATION".FIXTURE_1_STA_3_CALIB_MEM )
   END_RUNG
   // the same network as SCL:
   IF "DB4000_FIX_TABLE_POSITIONS".UNIT_01.FIXTURE_1.IN_CLADDING_STATION_3 AND "DB2031_CYCLES_GENERAL".CALIBRATION_CYCLE.CYCLE_SELECTED AND "DB2430_FULL_DEPTH".FD_UNIT_01.FIXTURE_1.FULL_DEPTH_STA_3 THEN
       "DB4001_FIXTURES_CALIBRATION".FIXTURE_1_STA_3_CALIB_MEM := TRUE;
   END_IF;
END_REGION

REGION Network 3: FIXTURE 2 STATION 2 CALIBRATION DONE MEMORY
   RUNG wire#powerrail
      Contact( "DB4000_FIX_TABLE_POSITIONS".UNIT_01.FIXTURE_2.IN_SPARE_STATION_2 )
      Contact( "DB2031_CYCLES_GENERAL".CALIBRATION_CYCLE.CYCLE_SELECTED )
      Contact( "DB2430_FULL_DEPTH".FD_UNIT_01.FIXTURE_2.FULL_DEPTH_STA_2 )
      S_Coil( "DB4001_FIXTURES_CALIBRATION".FIXTURE_2_STA_2_CALIB_MEM )
   END_RUNG
   // the same network as SCL:
   IF "DB4000_FIX_TABLE_POSITIONS".UNIT_01.FIXTURE_2.IN_SPARE_STATION_2 AND "DB2031_CYCLES_GENERAL".CALIBRATION_CYCLE.CYCLE_SELECTED AND "DB2430_FULL_DEPTH".FD_UNIT_01.FIXTURE_2.FULL_DEPTH_STA_2 THEN
       "DB4001_FIXTURES_CALIBRATION".FIXTURE_2_STA_2_CALIB_MEM := TRUE;
   END_IF;
END_REGION

REGION Network 4: FIXTURE 2 STATION 3 CALIBRATION MEMORY
   RUNG wire#powerrail
      Contact( "DB4000_FIX_TABLE_POSITIONS".UNIT_01.FIXTURE_2.IN_CLADDING_STATION_3 )
      Contact( "DB2031_CYCLES_GENERAL".CALIBRATION_CYCLE.CYCLE_SELECTED )
      Contact( "DB2430_FULL_DEPTH".FD_UNIT_01.FIXTURE_2.FULL_DEPTH_STA_3 )
      S_Coil( "DB4001_FIXTURES_CALIBRATION".FIXTURE_2_STA_3_CALIB_MEM )
   END_RUNG
   // the same network as SCL:
   IF "DB4000_FIX_TABLE_POSITIONS".UNIT_01.FIXTURE_2.IN_CLADDING_STATION_3 AND "DB2031_CYCLES_GENERAL".CALIBRATION_CYCLE.CYCLE_SELECTED AND "DB2430_FULL_DEPTH".FD_UNIT_01.FIXTURE_2.FULL_DEPTH_STA_3 THEN
       "DB4001_FIXTURES_CALIBRATION".FIXTURE_2_STA_3_CALIB_MEM := TRUE;
   END_IF;
END_REGION

REGION Network 5: FIXTURE 3 STATION 2 CALIBRATION DONE MEMORY
   RUNG wire#powerrail
      Contact( "DB4000_FIX_TABLE_POSITIONS".UNIT_01.FIXTURE_3.IN_SPARE_STATION_2 )
      Contact( "DB2031_CYCLES_GENERAL".CALIBRATION_CYCLE.CYCLE_SELECTED )
      Contact( "DB2430_FULL_DEPTH".FD_UNIT_01.FIXTURE_3.FULL_DEPTH_STA_2 )
      S_Coil( "DB4001_FIXTURES_CALIBRATION".FIXTURE_3_STA_2_CALIB_MEM )
   END_RUNG
   // the same network as SCL:
   IF "DB4000_FIX_TABLE_POSITIONS".UNIT_01.FIXTURE_3.IN_SPARE_STATION_2 AND "DB2031_CYCLES_GENERAL".CALIBRATION_CYCLE.CYCLE_SELECTED AND "DB2430_FULL_DEPTH".FD_UNIT_01.FIXTURE_3.FULL_DEPTH_STA_2 THEN
       "DB4001_FIXTURES_CALIBRATION".FIXTURE_3_STA_2_CALIB_MEM := TRUE;
   END_IF;
END_REGION

REGION Network 6: FIXTURE 3 STATION 3 CALIBRATION MEMORY
   RUNG wire#powerrail
      Contact( "DB4000_FIX_TABLE_POSITIONS".UNIT_01.FIXTURE_3.IN_CLADDING_STATION_3 )
      Contact( "DB2031_CYCLES_GENERAL".CALIBRATION_CYCLE.CYCLE_SELECTED )
      Contact( "DB2430_FULL_DEPTH".FD_UNIT_01.FIXTURE_3.FULL_DEPTH_STA_3 )
      S_Coil( "DB4001_FIXTURES_CALIBRATION".FIXTURE_3_STA_3_CALIB_MEM )
   END_RUNG
   // the same network as SCL:
   IF "DB4000_FIX_TABLE_POSITIONS".UNIT_01.FIXTURE_3.IN_CLADDING_STATION_3 AND "DB2031_CYCLES_GENERAL".CALIBRATION_CYCLE.CYCLE_SELECTED AND "DB2430_FULL_DEPTH".FD_UNIT_01.FIXTURE_3.FULL_DEPTH_STA_3 THEN
       "DB4001_FIXTURES_CALIBRATION".FIXTURE_3_STA_3_CALIB_MEM := TRUE;
   END_IF;
END_REGION

REGION Network 7: FIXTURE 4 STATION 2 CALIBRATION DONE MEMORY
   RUNG wire#powerrail
      Contact( "DB4000_FIX_TABLE_POSITIONS".UNIT_01.FIXTURE_4.IN_SPARE_STATION_2 )
      Contact( "DB2031_CYCLES_GENERAL".CALIBRATION_CYCLE.CYCLE_SELECTED )
      Contact( "DB2430_FULL_DEPTH".FD_UNIT_01.FIXTURE_4.FULL_DEPTH_STA_2 )
      S_Coil( "DB4001_FIXTURES_CALIBRATION".FIXTURE_4_STA_2_CALIB_MEM )
   END_RUNG
   // the same network as SCL:
   IF "DB4000_FIX_TABLE_POSITIONS".UNIT_01.FIXTURE_4.IN_SPARE_STATION_2 AND "DB2031_CYCLES_GENERAL".CALIBRATION_CYCLE.CYCLE_SELECTED AND "DB2430_FULL_DEPTH".FD_UNIT_01.FIXTURE_4.FULL_DEPTH_STA_2 THEN
       "DB4001_FIXTURES_CALIBRATION".FIXTURE_4_STA_2_CALIB_MEM := TRUE;
   END_IF;
END_REGION

REGION Network 8: FIXTURE 4 STATION 3 CALIBRATION MEMORY
   RUNG wire#powerrail
      Contact( "DB4000_FIX_TABLE_POSITIONS".UNIT_01.FIXTURE_4.IN_CLADDING_STATION_3 )
      Contact( "DB2031_CYCLES_GENERAL".CALIBRATION_CYCLE.CYCLE_SELECTED )
      Contact( "DB2430_FULL_DEPTH".FD_UNIT_01.FIXTURE_4.FULL_DEPTH_STA_3 )
      S_Coil( "DB4001_FIXTURES_CALIBRATION".FIXTURE_4_STA_3_CALIB_MEM )
   END_RUNG
   // the same network as SCL:
   IF "DB4000_FIX_TABLE_POSITIONS".UNIT_01.FIXTURE_4.IN_CLADDING_STATION_3 AND "DB2031_CYCLES_GENERAL".CALIBRATION_CYCLE.CYCLE_SELECTED AND "DB2430_FULL_DEPTH".FD_UNIT_01.FIXTURE_4.FULL_DEPTH_STA_3 THEN
       "DB4001_FIXTURES_CALIBRATION".FIXTURE_4_STA_3_CALIB_MEM := TRUE;
   END_IF;
END_REGION

REGION Network 9: ALL FIXTURES STATION 2 DONE
   RUNG wire#powerrail
      Contact( "DB4001_FIXTURES_CALIBRATION".FIXTURE_1_STA_2_CALIB_MEM )
      Contact( "DB4001_FIXTURES_CALIBRATION".FIXTURE_2_STA_2_CALIB_MEM )
      Contact( "DB4001_FIXTURES_CALIBRATION".FIXTURE_3_STA_2_CALIB_MEM )
      Contact( "DB4001_FIXTURES_CALIBRATION".FIXTURE_4_STA_2_CALIB_MEM )
      Coil( "DB4001_FIXTURES_CALIBRATION".ALL_FIXTURES_STA_2_CALIB_MEM )
   END_RUNG
   // the same network as SCL:
   "DB4001_FIXTURES_CALIBRATION".ALL_FIXTURES_STA_2_CALIB_MEM := "DB4001_FIXTURES_CALIBRATION".FIXTURE_1_STA_2_CALIB_MEM AND "DB4001_FIXTURES_CALIBRATION".FIXTURE_2_STA_2_CALIB_MEM AND "DB4001_FIXTURES_CALIBRATION".FIXTURE_3_STA_2_CALIB_MEM AND "DB4001_FIXTURES_CALIBRATION".FIXTURE_4_STA_2_CALIB_MEM;
END_REGION

REGION Network 10: ALL FIXTURES STATION 3 DONE
   RUNG wire#powerrail
      Contact( "DB4001_FIXTURES_CALIBRATION".FIXTURE_1_STA_3_CALIB_MEM )
      Contact( "DB4001_FIXTURES_CALIBRATION".FIXTURE_2_STA_3_CALIB_MEM )
      Contact( "DB4001_FIXTURES_CALIBRATION".FIXTURE_3_STA_3_CALIB_MEM )
      Contact( "DB4001_FIXTURES_CALIBRATION".FIXTURE_4_STA_3_CALIB_MEM )
      Coil( "DB4001_FIXTURES_CALIBRATION".ALL_FIXTURES_STA_3_CALIB_MEM )
   END_RUNG
   // the same network as SCL:
   "DB4001_FIXTURES_CALIBRATION".ALL_FIXTURES_STA_3_CALIB_MEM := "DB4001_FIXTURES_CALIBRATION".FIXTURE_1_STA_3_CALIB_MEM AND "DB4001_FIXTURES_CALIBRATION".FIXTURE_2_STA_3_CALIB_MEM AND "DB4001_FIXTURES_CALIBRATION".FIXTURE_3_STA_3_CALIB_MEM AND "DB4001_FIXTURES_CALIBRATION".FIXTURE_4_STA_3_CALIB_MEM;
END_REGION

REGION Network 11: ALL FIXTURES ALL STATIONS DONE
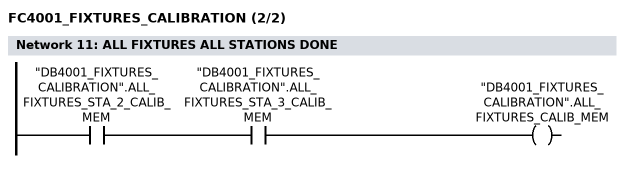
   RUNG wire#powerrail
      Contact( "DB4001_FIXTURES_CALIBRATION".ALL_FIXTURES_STA_2_CALIB_MEM )
      Contact( "DB4001_FIXTURES_CALIBRATION".ALL_FIXTURES_STA_3_CALIB_MEM )
      Coil( "DB4001_FIXTURES_CALIBRATION".ALL_FIXTURES_CALIB_MEM )
   END_RUNG
   // the same network as SCL:
   "DB4001_FIXTURES_CALIBRATION".ALL_FIXTURES_CALIB_MEM := "DB4001_FIXTURES_CALIBRATION".ALL_FIXTURES_STA_2_CALIB_MEM AND "DB4001_FIXTURES_CALIBRATION".ALL_FIXTURES_STA_3_CALIB_MEM;
END_REGION
END_FUNCTION

FUNCTION_BLOCK "FB2501_ANALOG_SENSOR"   // FB2501, LAD
{ S7_Optimized_Access := 'FALSE' }
AUTHOR : ETXETAR
VERSION : 1.0
// stored: AutoNumber false, IsIECCheckEnabled false, SetENOAutomatically false, UDAEnableTagReadback false
   VAR_INPUT
      INPUT : Word;   // INPUT
   END_VAR
   VAR_OUTPUT
      CLAMPED_WITHOUT_PART : Bool;   // CLAMPED WITHOUT PARTS / CLAMPED WITHOUT PART
      CLAMPED_WITH_PART : Bool;   // CLAMPED WITH PART
      CLAMPED_STATUS : Bool;   // CLAMPED / CLAMPED STATUS
      UNCLAMPED_STATUS : Bool;   // UNCLAMPED / UNCLAMPED STATUS
   END_VAR
   VAR DB_SPECIFIC
      CURRENT_VALUE { S7_SetPoint := 'True'} : DInt;   // CURRENT VALUE
      CLAMP_MAX_WITHOUT { S7_SetPoint := 'True'} : DInt;   // CLAMP MAX WITHOUT
      CLAMP_MIN_WITHOUT { S7_SetPoint := 'True'} : DInt := DINT#-10000;   // CLAMP MIN WITHOUT
      CLAMP_MAX_WITH { S7_SetPoint := 'True'} : DInt := DINT#-10000;   // CLAMP MAX WITH
      CLAMP_MIN_WITH { S7_SetPoint := 'True'} : DInt := DINT#-10000;   // CLAMP MIN WITH
      UNCLAMP_MAX { S7_SetPoint := 'True'} : DInt := DINT#-10000;   // UNCLAMP MAX
      UNCLAMP_MIN { S7_SetPoint := 'True'} : DInt := DINT#-10000;   // UNCLAMP MIN
      CLAMP_REQUEST { S7_SetPoint := 'True'} : Bool;   // CLAMP REQUEST
      UNCLAMP_REQUEST { S7_SetPoint := 'True'} : Bool;   // UNCLAMP REQUEST
      RELEASE_PRESSURE_REQUEST { S7_SetPoint := 'True'} : Bool;   // PRESSURE RELEASE REQUEST
   END_VAR
BEGIN

REGION Network 1: INPUTS
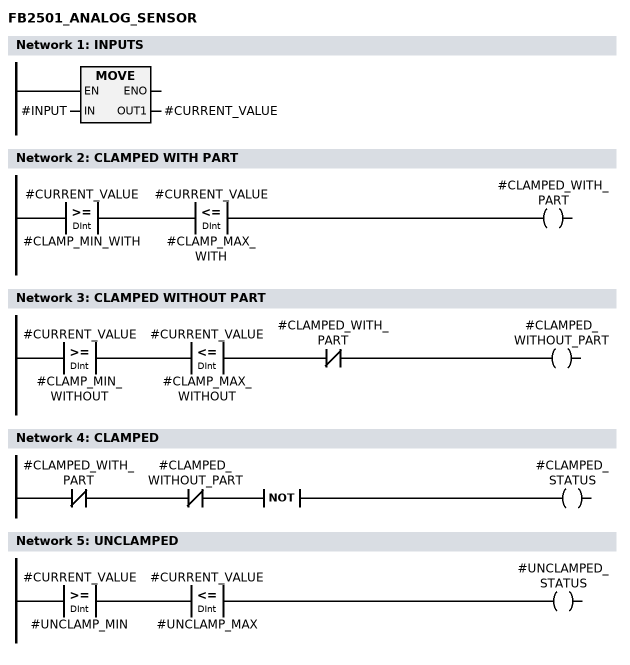
   RUNG wire#powerrail
      { S7_GenerateENO := "TRUE" } Move(in := #INPUT, out1 => #CURRENT_VALUE)
   END_RUNG
   // the same network as SCL:
   #CURRENT_VALUE := #INPUT;
END_REGION

REGION Network 2: CLAMPED WITH PART
   RUNG wire#powerrail
      { S7_Templates := "SrcType := DInt" } GE_Contact(in1 := #CURRENT_VALUE, in2 := #CLAMP_MIN_WITH)
      { S7_Templates := "SrcType := DInt" } LE_Contact(in1 := #CURRENT_VALUE, in2 := #CLAMP_MAX_WITH)
      Coil( #CLAMPED_WITH_PART )
   END_RUNG
   // the same network as SCL:
   #CLAMPED_WITH_PART := (#CURRENT_VALUE >= #CLAMP_MIN_WITH) AND (#CURRENT_VALUE <= #CLAMP_MAX_WITH);
END_REGION

REGION Network 3: CLAMPED WITHOUT PART
   RUNG wire#powerrail
      { S7_Templates := "SrcType := DInt" } GE_Contact(in1 := #CURRENT_VALUE, in2 := #CLAMP_MIN_WITHOUT)
      { S7_Templates := "SrcType := DInt" } LE_Contact(in1 := #CURRENT_VALUE, in2 := #CLAMP_MAX_WITHOUT)
      I_Contact( #CLAMPED_WITH_PART )
      Coil( #CLAMPED_WITHOUT_PART )
   END_RUNG
   // the same network as SCL:
   #CLAMPED_WITHOUT_PART := (#CURRENT_VALUE >= #CLAMP_MIN_WITHOUT) AND (#CURRENT_VALUE <= #CLAMP_MAX_WITHOUT) AND NOT #CLAMPED_WITH_PART;
END_REGION

REGION Network 4: CLAMPED
   RUNG wire#powerrail
      I_Contact( #CLAMPED_WITH_PART )
      I_Contact( #CLAMPED_WITHOUT_PART )
      Not()
      Coil( #CLAMPED_STATUS )
   END_RUNG
   // the same network as SCL:
   #CLAMPED_STATUS := NOT (NOT #CLAMPED_WITH_PART AND NOT #CLAMPED_WITHOUT_PART);
END_REGION

REGION Network 5: UNCLAMPED
   RUNG wire#powerrail
      { S7_Templates := "SrcType := DInt" } GE_Contact(in1 := #CURRENT_VALUE, in2 := #UNCLAMP_MIN)
      { S7_Templates := "SrcType := DInt" } LE_Contact(in1 := #CURRENT_VALUE, in2 := #UNCLAMP_MAX)
      Coil( #UNCLAMPED_STATUS )
   END_RUNG
   // the same network as SCL:
   #UNCLAMPED_STATUS := (#CURRENT_VALUE >= #UNCLAMP_MIN) AND (#CURRENT_VALUE <= #UNCLAMP_MAX);
END_REGION
END_FUNCTION_BLOCK

FUNCTION_BLOCK "FB2502_PART_DETECTION_SENSOR"   // FB2502, LAD
{ S7_Optimized_Access := 'FALSE' }
AUTHOR : ETXETAR
VERSION : 1.0
// stored: AutoNumber false, IsIECCheckEnabled false, SetENOAutomatically false, UDAEnableTagReadback false
   VAR_INPUT
      INPUT : Word;   // INPUT
   END_VAR
   VAR_OUTPUT
      PART_PRESENT_FACE_A : Bool;   // CLAMPED WITHOUT PARTS / PART PRESENT FACE A UP
      PART_PRESENT_FACE_B : Bool;   // CLAMPED WITH PART / PART PRESENT FACE B UP
      PART_PRESENT : Bool;   // CLAMPED / PART_PRESENT
      NO_PART_PRESENT : Bool;   // UNCLAMPED / NO PART PRESENT
   END_VAR
   VAR DB_SPECIFIC
      CURRENT_VALUE { S7_SetPoint := 'True'} : DInt;   // CURRENT VALUE
      PART_FACE_A_PRESENT_MAX { S7_SetPoint := 'True'} : DInt;   // CLAMP MAX WITHOUT
      PART_FACE_A_PRESENT_MIN { S7_SetPoint := 'True'} : DInt := DINT#-10000;   // CLAMP MIN WITHOUT
      PART_FACE_B_PRESENT_MAX { S7_SetPoint := 'True'} : DInt := DINT#-10000;   // CLAMP MAX WITH
      PART_FACE_B_PRESENT_MIN { S7_SetPoint := 'True'} : DInt := DINT#-10000;   // CLAMP MIN WITH
      NO_PART_PRESENT_MAX { S7_SetPoint := 'True'} : DInt := DINT#-10000;   // UNCLAMP MAX
      NO_PART_PRESENT_MIN { S7_SetPoint := 'True'} : DInt := DINT#-10000;   // UNCLAMP MIN
   END_VAR
BEGIN

REGION Network 1: INPUTS
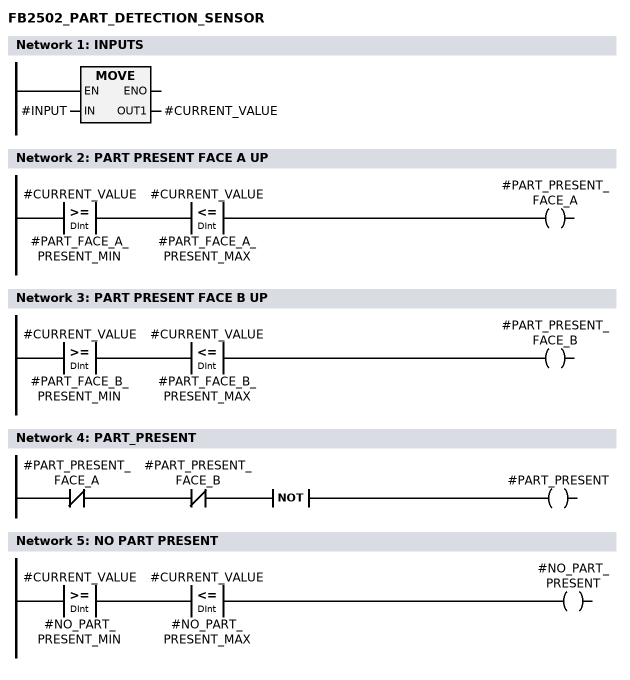
   RUNG wire#powerrail
      { S7_GenerateENO := "TRUE" } Move(in := #INPUT, out1 => #CURRENT_VALUE)
   END_RUNG
   // the same network as SCL:
   #CURRENT_VALUE := #INPUT;
END_REGION

REGION Network 2: PART PRESENT FACE A UP
   RUNG wire#powerrail
      { S7_Templates := "SrcType := DInt" } GE_Contact(in1 := #CURRENT_VALUE, in2 := #PART_FACE_A_PRESENT_MIN)
      { S7_Templates := "SrcType := DInt" } LE_Contact(in1 := #CURRENT_VALUE, in2 := #PART_FACE_A_PRESENT_MAX)
      Coil( #PART_PRESENT_FACE_A )
   END_RUNG
   // the same network as SCL:
   #PART_PRESENT_FACE_A := (#CURRENT_VALUE >= #PART_FACE_A_PRESENT_MIN) AND (#CURRENT_VALUE <= #PART_FACE_A_PRESENT_MAX);
END_REGION

REGION Network 3: PART PRESENT FACE B UP
   RUNG wire#powerrail
      { S7_Templates := "SrcType := DInt" } GE_Contact(in1 := #CURRENT_VALUE, in2 := #PART_FACE_B_PRESENT_MIN)
      { S7_Templates := "SrcType := DInt" } LE_Contact(in1 := #CURRENT_VALUE, in2 := #PART_FACE_B_PRESENT_MAX)
      Coil( #PART_PRESENT_FACE_B )
   END_RUNG
   // the same network as SCL:
   #PART_PRESENT_FACE_B := (#CURRENT_VALUE >= #PART_FACE_B_PRESENT_MIN) AND (#CURRENT_VALUE <= #PART_FACE_B_PRESENT_MAX);
END_REGION

REGION Network 4: PART_PRESENT
   RUNG wire#powerrail
      I_Contact( #PART_PRESENT_FACE_A )
      I_Contact( #PART_PRESENT_FACE_B )
      Not()
      Coil( #PART_PRESENT )
   END_RUNG
   // the same network as SCL:
   #PART_PRESENT := NOT (NOT #PART_PRESENT_FACE_A AND NOT #PART_PRESENT_FACE_B);
END_REGION

REGION Network 5: NO PART PRESENT
   RUNG wire#powerrail
      { S7_Templates := "SrcType := DInt" } GE_Contact(in1 := #CURRENT_VALUE, in2 := #NO_PART_PRESENT_MIN)
      { S7_Templates := "SrcType := DInt" } LE_Contact(in1 := #CURRENT_VALUE, in2 := #NO_PART_PRESENT_MAX)
      Coil( #NO_PART_PRESENT )
   END_RUNG
   // the same network as SCL:
   #NO_PART_PRESENT := (#CURRENT_VALUE >= #NO_PART_PRESENT_MIN) AND (#CURRENT_VALUE <= #NO_PART_PRESENT_MAX);
END_REGION
END_FUNCTION_BLOCK

FUNCTION "FC6500_CYLINDERS" : Void   // FC6500, LAD
{ S7_Optimized_Access := 'FALSE' }
AUTHOR : ETXETAR
VERSION : 1.0
// stored: AutoNumber false, IsIECCheckEnabled false, SetENOAutomatically false, UDAEnableTagReadback false
BEGIN

REGION Network 1: FC6600_UNIT_01_UP_SEALING_STRUCTURE
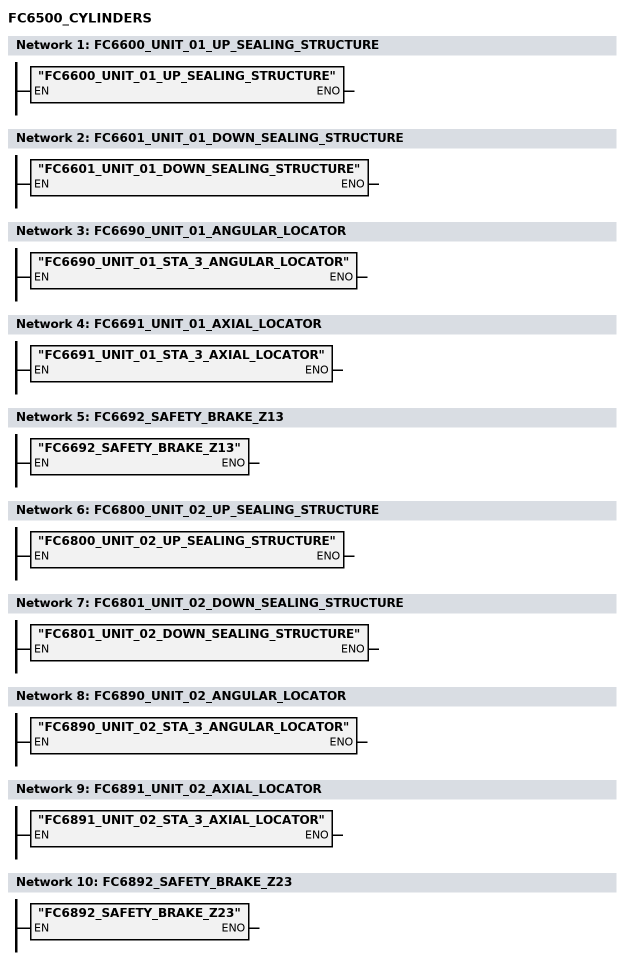
   RUNG wire#powerrail
      "FC6600_UNIT_01_UP_SEALING_STRUCTURE"()
   END_RUNG
   // the same network as SCL:
   "FC6600_UNIT_01_UP_SEALING_STRUCTURE"();
END_REGION

REGION Network 2: FC6601_UNIT_01_DOWN_SEALING_STRUCTURE
   RUNG wire#powerrail
      "FC6601_UNIT_01_DOWN_SEALING_STRUCTURE"()
   END_RUNG
   // the same network as SCL:
   "FC6601_UNIT_01_DOWN_SEALING_STRUCTURE"();
END_REGION

REGION Network 3: FC6690_UNIT_01_ANGULAR_LOCATOR
   RUNG wire#powerrail
      "FC6690_UNIT_01_STA_3_ANGULAR_LOCATOR"()
   END_RUNG
   // the same network as SCL:
   "FC6690_UNIT_01_STA_3_ANGULAR_LOCATOR"();
END_REGION

REGION Network 4: FC6691_UNIT_01_AXIAL_LOCATOR
   RUNG wire#powerrail
      "FC6691_UNIT_01_STA_3_AXIAL_LOCATOR"()
   END_RUNG
   // the same network as SCL:
   "FC6691_UNIT_01_STA_3_AXIAL_LOCATOR"();
END_REGION

REGION Network 5: FC6692_SAFETY_BRAKE_Z13
   RUNG wire#powerrail
      "FC6692_SAFETY_BRAKE_Z13"()
   END_RUNG
   // the same network as SCL:
   "FC6692_SAFETY_BRAKE_Z13"();
END_REGION

REGION Network 6: FC6800_UNIT_02_UP_SEALING_STRUCTURE
   RUNG wire#powerrail
      "FC6800_UNIT_02_UP_SEALING_STRUCTURE"()
   END_RUNG
   // the same network as SCL:
   "FC6800_UNIT_02_UP_SEALING_STRUCTURE"();
END_REGION

REGION Network 7: FC6801_UNIT_02_DOWN_SEALING_STRUCTURE
   RUNG wire#powerrail
      "FC6801_UNIT_02_DOWN_SEALING_STRUCTURE"()
   END_RUNG
   // the same network as SCL:
   "FC6801_UNIT_02_DOWN_SEALING_STRUCTURE"();
END_REGION

REGION Network 8: FC6890_UNIT_02_ANGULAR_LOCATOR
   RUNG wire#powerrail
      "FC6890_UNIT_02_STA_3_ANGULAR_LOCATOR"()
   END_RUNG
   // the same network as SCL:
   "FC6890_UNIT_02_STA_3_ANGULAR_LOCATOR"();
END_REGION

REGION Network 9: FC6891_UNIT_02_AXIAL_LOCATOR
   RUNG wire#powerrail
      "FC6891_UNIT_02_STA_3_AXIAL_LOCATOR"()
   END_RUNG
   // the same network as SCL:
   "FC6891_UNIT_02_STA_3_AXIAL_LOCATOR"();
END_REGION

REGION Network 10: FC6892_SAFETY_BRAKE_Z23
   RUNG wire#powerrail
      "FC6892_SAFETY_BRAKE_Z23"()
   END_RUNG
   // the same network as SCL:
   "FC6892_SAFETY_BRAKE_Z23"();
END_REGION
END_FUNCTION

FUNCTION "FC7000_SAFETY_DOORS" : Void   // FC7000, LAD
{ S7_Optimized_Access := 'FALSE' }
AUTHOR : ETXETAR
VERSION : 1.0
// stored: AutoNumber false, IsIECCheckEnabled false, SetENOAutomatically false, UDAEnableTagReadback false
BEGIN

REGION Network 1: CALL FC7002 UNIT 01 STATION 2 SAFETY DOOR
   // 2#0000_0001 OPTIONS 0 BIT 0 IMMEDIATE STOP REACTION OPTION
   // 2#0000_0010 OPTIONS 0 BIT 1 SEOC WARNING REACTION OPTION
   // 2#0000_0100 OPTIONS 0 BIT 2 CLOSED SENSOR INPUT OPTION
   // 2#0000_1000 OPTIONS 0 BIT 3 CIRCUIT E2 OPTION
   // 2#0001_0000 OPTIONS 0 BIT 4 HYDRAULIC DRIVE OPTION
   // 2#0010_0000 OPTIONS 0 BIT 5 CHIP CONVEYOR OPTION
   // 2#0100_0000 OPTIONS 0 BIT 6 SPARE OPTION
   // 2#1000_0000 OPTIONS 0 BIT 7 SPARE OPTION
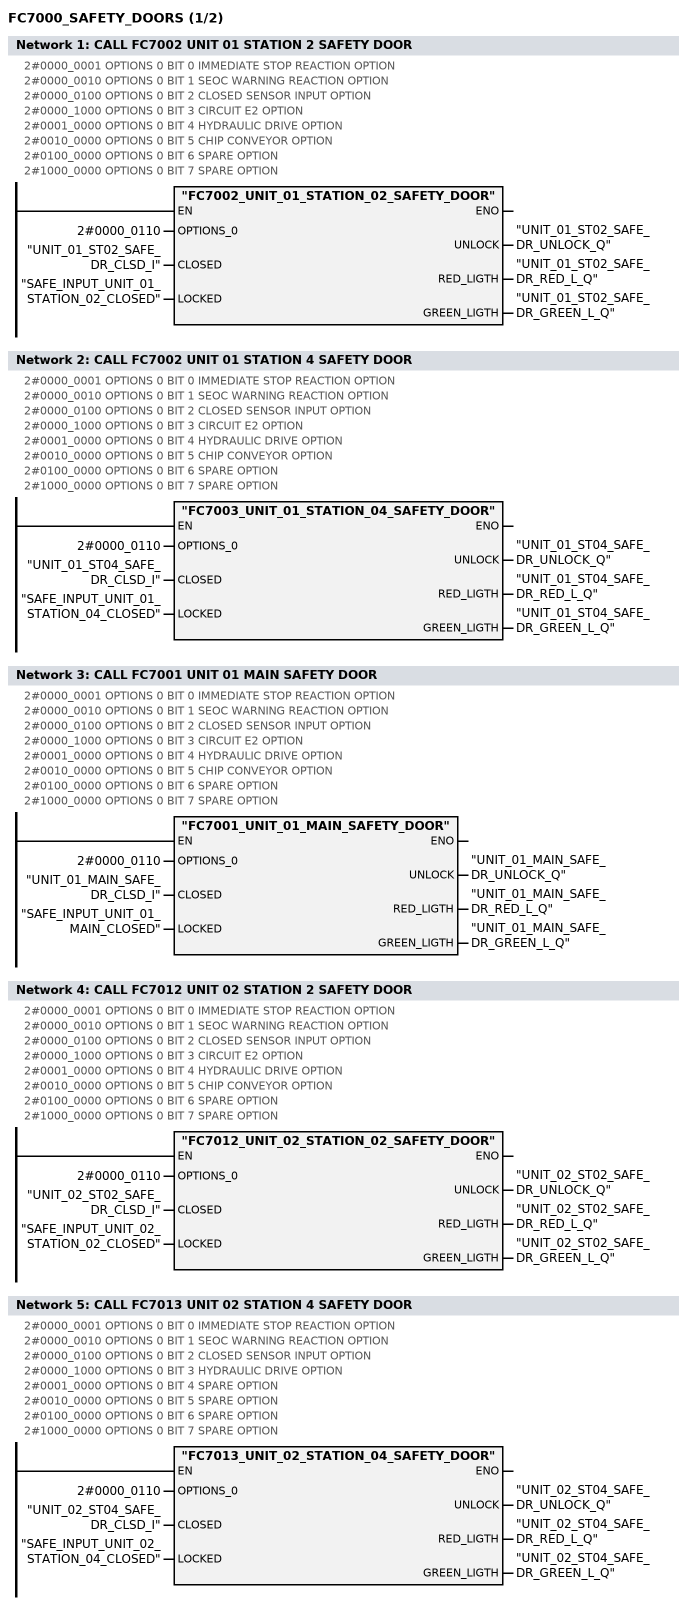
   RUNG wire#powerrail
      "FC7002_UNIT_01_STATION_02_SAFETY_DOOR"(OPTIONS_0 := 2#0000_0110, CLOSED := "UNIT_01_ST02_SAFE_DR_CLSD_I", LOCKED := "SAFE_INPUT_UNIT_01_STATION_02_CLOSED", UNLOCK => "UNIT_01_ST02_SAFE_DR_UNLOCK_Q", RED_LIGTH => "UNIT_01_ST02_SAFE_DR_RED_L_Q", GREEN_LIGTH => "UNIT_01_ST02_SAFE_DR_GREEN_L_Q")
   END_RUNG
   // the same network as SCL:
   "FC7002_UNIT_01_STATION_02_SAFETY_DOOR"(OPTIONS_0 := 2#0000_0110,
                           CLOSED := "UNIT_01_ST02_SAFE_DR_CLSD_I",
                           LOCKED := "SAFE_INPUT_UNIT_01_STATION_02_CLOSED",
                           UNLOCK => "UNIT_01_ST02_SAFE_DR_UNLOCK_Q",
                           RED_LIGTH => "UNIT_01_ST02_SAFE_DR_RED_L_Q",
                           GREEN_LIGTH => "UNIT_01_ST02_SAFE_DR_GREEN_L_Q");
END_REGION

REGION Network 2: CALL FC7002 UNIT 01 STATION 4 SAFETY DOOR
   // 2#0000_0001 OPTIONS 0 BIT 0 IMMEDIATE STOP REACTION OPTION
   // 2#0000_0010 OPTIONS 0 BIT 1 SEOC WARNING REACTION OPTION
   // 2#0000_0100 OPTIONS 0 BIT 2 CLOSED SENSOR INPUT OPTION
   // 2#0000_1000 OPTIONS 0 BIT 3 CIRCUIT E2 OPTION
   // 2#0001_0000 OPTIONS 0 BIT 4 HYDRAULIC DRIVE OPTION
   // 2#0010_0000 OPTIONS 0 BIT 5 CHIP CONVEYOR OPTION
   // 2#0100_0000 OPTIONS 0 BIT 6 SPARE OPTION
   // 2#1000_0000 OPTIONS 0 BIT 7 SPARE OPTION
   RUNG wire#powerrail
      "FC7003_UNIT_01_STATION_04_SAFETY_DOOR"(OPTIONS_0 := 2#0000_0110, CLOSED := "UNIT_01_ST04_SAFE_DR_CLSD_I", LOCKED := "SAFE_INPUT_UNIT_01_STATION_04_CLOSED", UNLOCK => "UNIT_01_ST04_SAFE_DR_UNLOCK_Q", RED_LIGTH => "UNIT_01_ST04_SAFE_DR_RED_L_Q", GREEN_LIGTH => "UNIT_01_ST04_SAFE_DR_GREEN_L_Q")
   END_RUNG
   // the same network as SCL:
   "FC7003_UNIT_01_STATION_04_SAFETY_DOOR"(OPTIONS_0 := 2#0000_0110,
                           CLOSED := "UNIT_01_ST04_SAFE_DR_CLSD_I",
                           LOCKED := "SAFE_INPUT_UNIT_01_STATION_04_CLOSED",
                           UNLOCK => "UNIT_01_ST04_SAFE_DR_UNLOCK_Q",
                           RED_LIGTH => "UNIT_01_ST04_SAFE_DR_RED_L_Q",
                           GREEN_LIGTH => "UNIT_01_ST04_SAFE_DR_GREEN_L_Q");
END_REGION

REGION Network 3: CALL FC7001 UNIT 01 MAIN SAFETY DOOR
   // 2#0000_0001 OPTIONS 0 BIT 0 IMMEDIATE STOP REACTION OPTION
   // 2#0000_0010 OPTIONS 0 BIT 1 SEOC WARNING REACTION OPTION
   // 2#0000_0100 OPTIONS 0 BIT 2 CLOSED SENSOR INPUT OPTION
   // 2#0000_1000 OPTIONS 0 BIT 3 CIRCUIT E2 OPTION
   // 2#0001_0000 OPTIONS 0 BIT 4 HYDRAULIC DRIVE OPTION
   // 2#0010_0000 OPTIONS 0 BIT 5 CHIP CONVEYOR OPTION
   // 2#0100_0000 OPTIONS 0 BIT 6 SPARE OPTION
   // 2#1000_0000 OPTIONS 0 BIT 7 SPARE OPTION
   RUNG wire#powerrail
      "FC7001_UNIT_01_MAIN_SAFETY_DOOR"(OPTIONS_0 := 2#0000_0110, CLOSED := "UNIT_01_MAIN_SAFE_DR_CLSD_I", LOCKED := "SAFE_INPUT_UNIT_01_MAIN_CLOSED", UNLOCK => "UNIT_01_MAIN_SAFE_DR_UNLOCK_Q", RED_LIGTH => "UNIT_01_MAIN_SAFE_DR_RED_L_Q", GREEN_LIGTH => "UNIT_01_MAIN_SAFE_DR_GREEN_L_Q")
   END_RUNG
   // the same network as SCL:
   "FC7001_UNIT_01_MAIN_SAFETY_DOOR"(OPTIONS_0 := 2#0000_0110,
                           CLOSED := "UNIT_01_MAIN_SAFE_DR_CLSD_I",
                           LOCKED := "SAFE_INPUT_UNIT_01_MAIN_CLOSED",
                           UNLOCK => "UNIT_01_MAIN_SAFE_DR_UNLOCK_Q",
                           RED_LIGTH => "UNIT_01_MAIN_SAFE_DR_RED_L_Q",
                           GREEN_LIGTH => "UNIT_01_MAIN_SAFE_DR_GREEN_L_Q");
END_REGION

REGION Network 4: CALL FC7012 UNIT 02 STATION 2 SAFETY DOOR
   // 2#0000_0001 OPTIONS 0 BIT 0 IMMEDIATE STOP REACTION OPTION
   // 2#0000_0010 OPTIONS 0 BIT 1 SEOC WARNING REACTION OPTION
   // 2#0000_0100 OPTIONS 0 BIT 2 CLOSED SENSOR INPUT OPTION
   // 2#0000_1000 OPTIONS 0 BIT 3 CIRCUIT E2 OPTION
   // 2#0001_0000 OPTIONS 0 BIT 4 HYDRAULIC DRIVE OPTION
   // 2#0010_0000 OPTIONS 0 BIT 5 CHIP CONVEYOR OPTION
   // 2#0100_0000 OPTIONS 0 BIT 6 SPARE OPTION
   // 2#1000_0000 OPTIONS 0 BIT 7 SPARE OPTION
   RUNG wire#powerrail
      "FC7012_UNIT_02_STATION_02_SAFETY_DOOR"(OPTIONS_0 := 2#0000_0110, CLOSED := "UNIT_02_ST02_SAFE_DR_CLSD_I", LOCKED := "SAFE_INPUT_UNIT_02_STATION_02_CLOSED", UNLOCK => "UNIT_02_ST02_SAFE_DR_UNLOCK_Q", RED_LIGTH => "UNIT_02_ST02_SAFE_DR_RED_L_Q", GREEN_LIGTH => "UNIT_02_ST02_SAFE_DR_GREEN_L_Q")
   END_RUNG
   // the same network as SCL:
   "FC7012_UNIT_02_STATION_02_SAFETY_DOOR"(OPTIONS_0 := 2#0000_0110,
                           CLOSED := "UNIT_02_ST02_SAFE_DR_CLSD_I",
                           LOCKED := "SAFE_INPUT_UNIT_02_STATION_02_CLOSED",
                           UNLOCK => "UNIT_02_ST02_SAFE_DR_UNLOCK_Q",
                           RED_LIGTH => "UNIT_02_ST02_SAFE_DR_RED_L_Q",
                           GREEN_LIGTH => "UNIT_02_ST02_SAFE_DR_GREEN_L_Q");
END_REGION

REGION Network 5: CALL FC7013 UNIT 02 STATION 4 SAFETY DOOR
   // 2#0000_0001 OPTIONS 0 BIT 0 IMMEDIATE STOP REACTION OPTION
   // 2#0000_0010 OPTIONS 0 BIT 1 SEOC WARNING REACTION OPTION
   // 2#0000_0100 OPTIONS 0 BIT 2 CLOSED SENSOR INPUT OPTION
   // 2#0000_1000 OPTIONS 0 BIT 3 HYDRAULIC DRIVE OPTION
   // 2#0001_0000 OPTIONS 0 BIT 4 SPARE OPTION
   // 2#0010_0000 OPTIONS 0 BIT 5 SPARE OPTION
   // 2#0100_0000 OPTIONS 0 BIT 6 SPARE OPTION
   // 2#1000_0000 OPTIONS 0 BIT 7 SPARE OPTION
   RUNG wire#powerrail
      "FC7013_UNIT_02_STATION_04_SAFETY_DOOR"(OPTIONS_0 := 2#0000_0110, CLOSED := "UNIT_02_ST04_SAFE_DR_CLSD_I", LOCKED := "SAFE_INPUT_UNIT_02_STATION_04_CLOSED", UNLOCK => "UNIT_02_ST04_SAFE_DR_UNLOCK_Q", RED_LIGTH => "UNIT_02_ST04_SAFE_DR_RED_L_Q", GREEN_LIGTH => "UNIT_02_ST04_SAFE_DR_GREEN_L_Q")
   END_RUNG
   // the same network as SCL:
   "FC7013_UNIT_02_STATION_04_SAFETY_DOOR"(OPTIONS_0 := 2#0000_0110,
                           CLOSED := "UNIT_02_ST04_SAFE_DR_CLSD_I",
                           LOCKED := "SAFE_INPUT_UNIT_02_STATION_04_CLOSED",
                           UNLOCK => "UNIT_02_ST04_SAFE_DR_UNLOCK_Q",
                           RED_LIGTH => "UNIT_02_ST04_SAFE_DR_RED_L_Q",
                           GREEN_LIGTH => "UNIT_02_ST04_SAFE_DR_GREEN_L_Q");
END_REGION

REGION Network 6: CALL FC7011 UNIT 02 MAIN SAFETY DOOR
   // 2#0000_0001 OPTIONS 0 BIT 0 IMMEDIATE STOP REACTION OPTION
   // 2#0000_0010 OPTIONS 0 BIT 1 SEOC WARNING REACTION OPTION
   // 2#0000_0100 OPTIONS 0 BIT 2 CLOSED SENSOR INPUT OPTION
   // 2#0000_1000 OPTIONS 0 BIT 3 CIRCUIT E2 OPTION
   // 2#0001_0000 OPTIONS 0 BIT 4 HYDRAULIC DRIVE OPTION
   // 2#0010_0000 OPTIONS 0 BIT 5 CHIP CONVEYOR OPTION
   // 2#0100_0000 OPTIONS 0 BIT 6 SPARE OPTION
   // 2#1000_0000 OPTIONS 0 BIT 7 SPARE OPTION
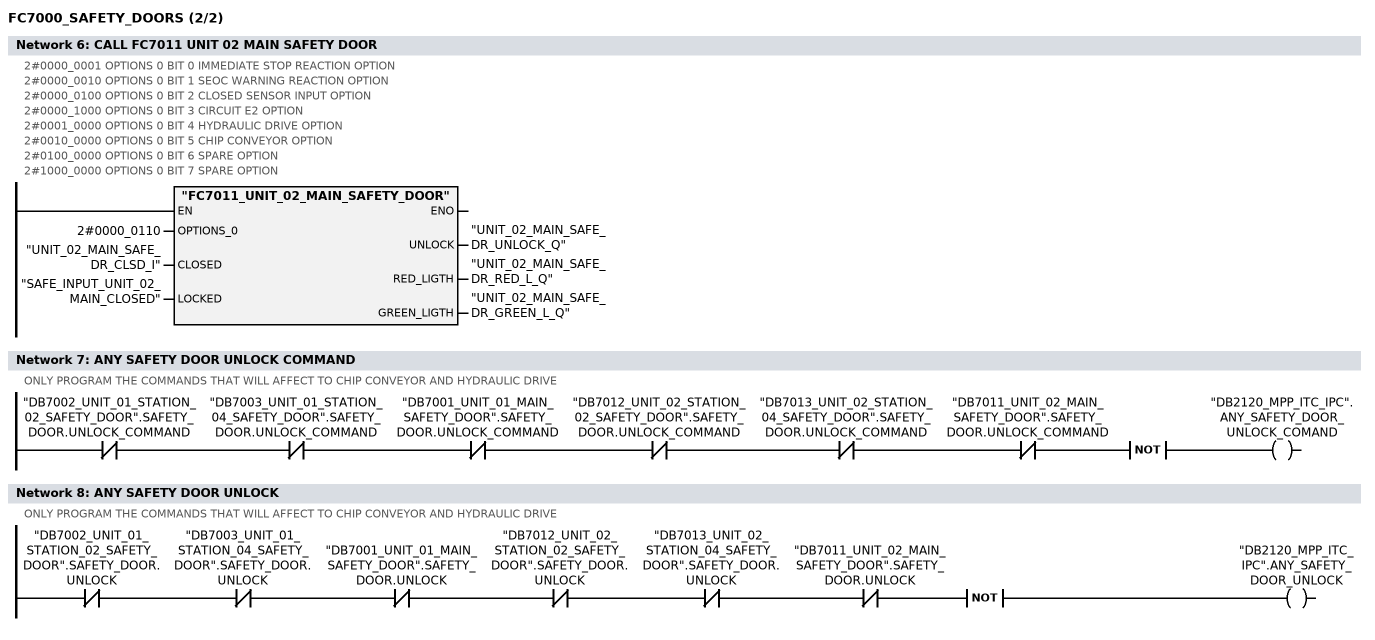
   RUNG wire#powerrail
      "FC7011_UNIT_02_MAIN_SAFETY_DOOR"(OPTIONS_0 := 2#0000_0110, CLOSED := "UNIT_02_MAIN_SAFE_DR_CLSD_I", LOCKED := "SAFE_INPUT_UNIT_02_MAIN_CLOSED", UNLOCK => "UNIT_02_MAIN_SAFE_DR_UNLOCK_Q", RED_LIGTH => "UNIT_02_MAIN_SAFE_DR_RED_L_Q", GREEN_LIGTH => "UNIT_02_MAIN_SAFE_DR_GREEN_L_Q")
   END_RUNG
   // the same network as SCL:
   "FC7011_UNIT_02_MAIN_SAFETY_DOOR"(OPTIONS_0 := 2#0000_0110,
                           CLOSED := "UNIT_02_MAIN_SAFE_DR_CLSD_I",
                           LOCKED := "SAFE_INPUT_UNIT_02_MAIN_CLOSED",
                           UNLOCK => "UNIT_02_MAIN_SAFE_DR_UNLOCK_Q",
                           RED_LIGTH => "UNIT_02_MAIN_SAFE_DR_RED_L_Q",
                           GREEN_LIGTH => "UNIT_02_MAIN_SAFE_DR_GREEN_L_Q");
END_REGION

REGION Network 7: ANY SAFETY DOOR UNLOCK COMMAND
   // ONLY PROGRAM THE COMMANDS THAT WILL AFFECT TO CHIP CONVEYOR AND HYDRAULIC DRIVE
   RUNG wire#powerrail
      I_Contact( "DB7002_UNIT_01_STATION_02_SAFETY_DOOR".SAFETY_DOOR.UNLOCK_COMMAND )
      I_Contact( "DB7003_UNIT_01_STATION_04_SAFETY_DOOR".SAFETY_DOOR.UNLOCK_COMMAND )
      I_Contact( "DB7001_UNIT_01_MAIN_SAFETY_DOOR".SAFETY_DOOR.UNLOCK_COMMAND )
      I_Contact( "DB7012_UNIT_02_STATION_02_SAFETY_DOOR".SAFETY_DOOR.UNLOCK_COMMAND )
      I_Contact( "DB7013_UNIT_02_STATION_04_SAFETY_DOOR".SAFETY_DOOR.UNLOCK_COMMAND )
      I_Contact( "DB7011_UNIT_02_MAIN_SAFETY_DOOR".SAFETY_DOOR.UNLOCK_COMMAND )
      Not()
      Coil( "DB2120_MPP_ITC_IPC".ANY_SAFETY_DOOR_UNLOCK_COMAND )
   END_RUNG
   // the same network as SCL:
   "DB2120_MPP_ITC_IPC".ANY_SAFETY_DOOR_UNLOCK_COMAND := NOT (NOT "DB7002_UNIT_01_STATION_02_SAFETY_DOOR".SAFETY_DOOR.UNLOCK_COMMAND AND NOT "DB7003_UNIT_01_STATION_04_SAFETY_DOOR".SAFETY_DOOR.UNLOCK_COMMAND AND NOT "DB7001_UNIT_01_MAIN_SAFETY_DOOR".SAFETY_DOOR.UNLOCK_COMMAND AND NOT "DB7012_UNIT_02_STATION_02_SAFETY_DOOR".SAFETY_DOOR.UNLOCK_COMMAND AND NOT "DB7013_UNIT_02_STATION_04_SAFETY_DOOR".SAFETY_DOOR.UNLOCK_COMMAND AND NOT "DB7011_UNIT_02_MAIN_SAFETY_DOOR".SAFETY_DOOR.UNLOCK_COMMAND);
END_REGION

REGION Network 8: ANY SAFETY DOOR UNLOCK
   // ONLY PROGRAM THE COMMANDS THAT WILL AFFECT TO CHIP CONVEYOR AND HYDRAULIC DRIVE
   RUNG wire#powerrail
      I_Contact( "DB7002_UNIT_01_STATION_02_SAFETY_DOOR".SAFETY_DOOR.UNLOCK )
      I_Contact( "DB7003_UNIT_01_STATION_04_SAFETY_DOOR".SAFETY_DOOR.UNLOCK )
      I_Contact( "DB7001_UNIT_01_MAIN_SAFETY_DOOR".SAFETY_DOOR.UNLOCK )
      I_Contact( "DB7012_UNIT_02_STATION_02_SAFETY_DOOR".SAFETY_DOOR.UNLOCK )
      I_Contact( "DB7013_UNIT_02_STATION_04_SAFETY_DOOR".SAFETY_DOOR.UNLOCK )
      I_Contact( "DB7011_UNIT_02_MAIN_SAFETY_DOOR".SAFETY_DOOR.UNLOCK )
      Not()
      Coil( "DB2120_MPP_ITC_IPC".ANY_SAFETY_DOOR_UNLOCK )
   END_RUNG
   // the same network as SCL:
   "DB2120_MPP_ITC_IPC".ANY_SAFETY_DOOR_UNLOCK := NOT (NOT "DB7002_UNIT_01_STATION_02_SAFETY_DOOR".SAFETY_DOOR.UNLOCK AND NOT "DB7003_UNIT_01_STATION_04_SAFETY_DOOR".SAFETY_DOOR.UNLOCK AND NOT "DB7001_UNIT_01_MAIN_SAFETY_DOOR".SAFETY_DOOR.UNLOCK AND NOT "DB7012_UNIT_02_STATION_02_SAFETY_DOOR".SAFETY_DOOR.UNLOCK AND NOT "DB7013_UNIT_02_STATION_04_SAFETY_DOOR".SAFETY_DOOR.UNLOCK AND NOT "DB7011_UNIT_02_MAIN_SAFETY_DOOR".SAFETY_DOOR.UNLOCK);
END_REGION
END_FUNCTION

FUNCTION "FC7200_HMI_FUNCTION" : Void   // FC7200, LAD
{ S7_Optimized_Access := 'FALSE' }
AUTHOR : ETXETAR
VERSION : 1.0
// stored: AutoNumber false, IsIECCheckEnabled false, SetENOAutomatically false, UDAEnableTagReadback false
   VAR_TEMP
      SCREEN_NAV : Bool;   // SCREEN NAVEGATION OPTION
      CNC_STATUS : Bool;   // CNC STATUS OPTION
      X : Int;
   END_VAR
   VAR CONSTANT
      TOTAL_SCREEN_NUM : Int := 89;
      FC_NUMBER : DInt := 7200;
   END_VAR
BEGIN

REGION Network 1: OPTIONS OFF
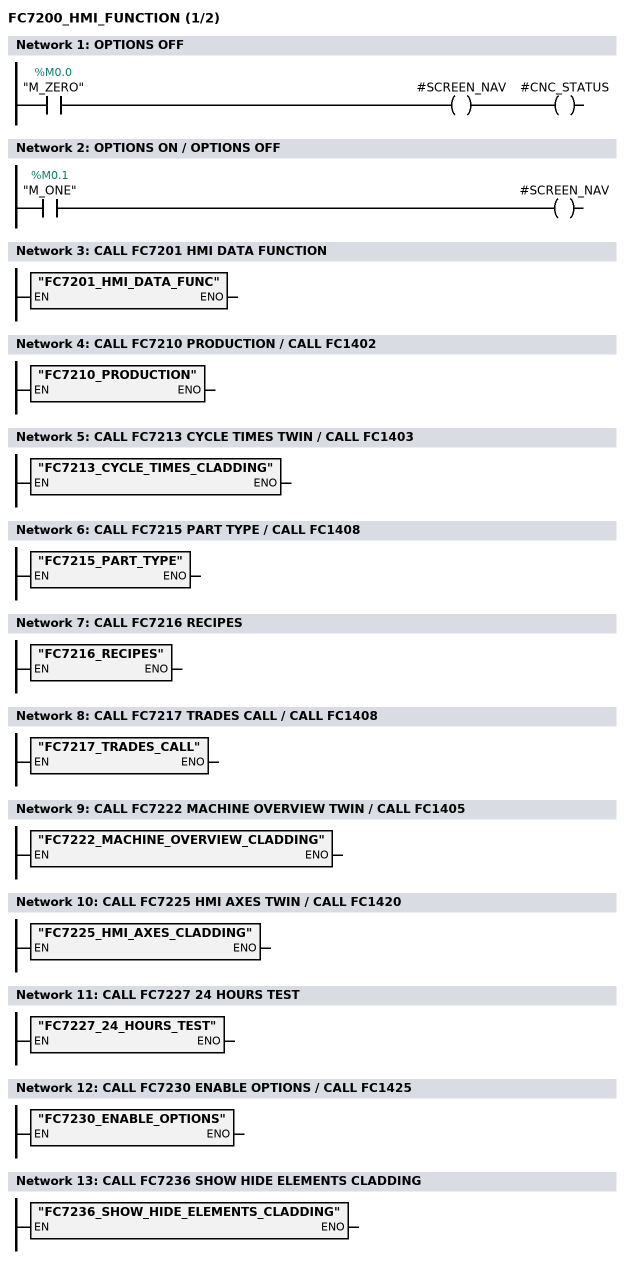
   RUNG wire#powerrail
      Contact( "M_ZERO" )
      Coil( #SCREEN_NAV )
      Coil( #CNC_STATUS )
   END_RUNG
   // the same network as SCL:
   #SCREEN_NAV := "M_ZERO";
   #CNC_STATUS := "M_ZERO";
END_REGION

REGION Network 2: OPTIONS ON / OPTIONS OFF
   RUNG wire#powerrail
      Contact( "M_ONE" )
      Coil( #SCREEN_NAV )
   END_RUNG
   // the same network as SCL:
   #SCREEN_NAV := "M_ONE";
END_REGION

REGION Network 3: CALL FC7201 HMI DATA FUNCTION
   RUNG wire#powerrail
      "FC7201_HMI_DATA_FUNC"()
   END_RUNG
   // the same network as SCL:
   "FC7201_HMI_DATA_FUNC"();
END_REGION

REGION Network 4: CALL FC7210 PRODUCTION / CALL FC1402
   RUNG wire#powerrail
      "FC7210_PRODUCTION"()
   END_RUNG
   // the same network as SCL:
   "FC7210_PRODUCTION"();
END_REGION

REGION Network 5: CALL FC7213 CYCLE TIMES TWIN / CALL FC1403
   RUNG wire#powerrail
      "FC7213_CYCLE_TIMES_CLADDING"()
   END_RUNG
   // the same network as SCL:
   "FC7213_CYCLE_TIMES_CLADDING"();
END_REGION

REGION Network 6: CALL FC7215 PART TYPE / CALL FC1408
   RUNG wire#powerrail
      "FC7215_PART_TYPE"()
   END_RUNG
   // the same network as SCL:
   "FC7215_PART_TYPE"();
END_REGION

REGION Network 7: CALL FC7216 RECIPES
   RUNG wire#powerrail
      "FC7216_RECIPES"()
   END_RUNG
   // the same network as SCL:
   "FC7216_RECIPES"();
END_REGION

REGION Network 8: CALL FC7217 TRADES CALL / CALL FC1408
   RUNG wire#powerrail
      "FC7217_TRADES_CALL"()
   END_RUNG
   // the same network as SCL:
   "FC7217_TRADES_CALL"();
END_REGION

REGION Network 9: CALL FC7222 MACHINE OVERVIEW TWIN / CALL FC1405
   RUNG wire#powerrail
      "FC7222_MACHINE_OVERVIEW_CLADDING"()
   END_RUNG
   // the same network as SCL:
   "FC7222_MACHINE_OVERVIEW_CLADDING"();
END_REGION

REGION Network 10: CALL FC7225 HMI AXES TWIN / CALL FC1420
   RUNG wire#powerrail
      "FC7225_HMI_AXES_CLADDING"()
   END_RUNG
   // the same network as SCL:
   "FC7225_HMI_AXES_CLADDING"();
END_REGION

REGION Network 11: CALL FC7227 24 HOURS TEST
   RUNG wire#powerrail
      "FC7227_24_HOURS_TEST"()
   END_RUNG
   // the same network as SCL:
   "FC7227_24_HOURS_TEST"();
END_REGION

REGION Network 12: CALL FC7230 ENABLE OPTIONS / CALL FC1425
   RUNG wire#powerrail
      "FC7230_ENABLE_OPTIONS"()
   END_RUNG
   // the same network as SCL:
   "FC7230_ENABLE_OPTIONS"();
END_REGION

REGION Network 13: CALL FC7236 SHOW HIDE ELEMENTS CLADDING
   RUNG wire#powerrail
      "FC7236_SHOW_HIDE_ELEMENTS_CLADDING"()
   END_RUNG
   // the same network as SCL:
   "FC7236_SHOW_HIDE_ELEMENTS_CLADDING"();
END_REGION

REGION Network 14 (SCL): SCREEN NAVIGATION

       IF #SCREEN_NAV THEN
           FOR #X := 11 TO #TOTAL_SCREEN_NUM DO
               IF "DB7200_HMI_FUNCTION".SCREEN_SELECTION[#X] THEN
                   "DB7200_HMI_FUNCTION".PLC_SCREEN_SELECTION :=INT_TO_WORD(#X);
               END_IF;
           END_FOR;
       END_IF;
END_REGION

REGION Network 15: CNC STATUS
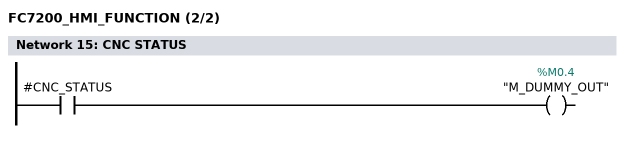
   RUNG wire#powerrail
      Contact( #CNC_STATUS )
      Coil( "M_DUMMY_OUT" )
   END_RUNG
   // the same network as SCL:
   "M_DUMMY_OUT" := #CNC_STATUS;
END_REGION
END_FUNCTION

FUNCTION "FC8007_UNIT_03_PART_STATUS_FULL_DEPTH" : Void   // FC8007, LAD
{ S7_Optimized_Access := 'TRUE' }
VERSION : 0.1
// stored: AutoNumber false, IsIECCheckEnabled false, SetENOAutomatically false, UDAEnableTagReadback false
BEGIN

REGION Network 1: FIXTURE 1 PART STATUS UNIT 01
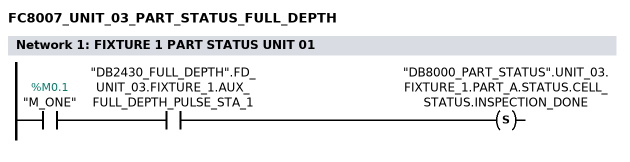
   RUNG wire#powerrail
      Contact( "M_ONE" )
      Contact( "DB2430_FULL_DEPTH".FD_UNIT_03.FIXTURE_1.AUX_FULL_DEPTH_PULSE_STA_1 )
      S_Coil( "DB8000_PART_STATUS".UNIT_03.FIXTURE_1.PART_A.STATUS.CELL_STATUS.INSPECTION_DONE )
   END_RUNG
   // the same network as SCL:
   IF "M_ONE" AND "DB2430_FULL_DEPTH".FD_UNIT_03.FIXTURE_1.AUX_FULL_DEPTH_PULSE_STA_1 THEN
       "DB8000_PART_STATUS".UNIT_03.FIXTURE_1.PART_A.STATUS.CELL_STATUS.INSPECTION_DONE := TRUE;
   END_IF;
END_REGION
END_FUNCTION

DATA_BLOCK "DB21205_UNIT_01_COMBINER_MEDICOAT"   // DB21205
{ DB_Accessible_From_OPC_UA := 'FALSE' }
VERSION : 0.1
// stored: AutoNumber false, DBAccessibleFromOPCUA false, DBAccessibleFromWebserver true, InstanceOfName FB21200_POWDER_FLOW_SENSOR_MEDICOAT, InstanceOfType FB
"FB21200_POWDER_FLOW_SENSOR_MEDICOAT"
BEGIN
END_DATA_BLOCK

DATA_BLOCK "DB21206_UNIT_02_COMBINER_MEDICOAT"   // DB21206
{ DB_Accessible_From_OPC_UA := 'FALSE' }
VERSION : 0.1
// stored: AutoNumber false, DBAccessibleFromOPCUA false, DBAccessibleFromWebserver true, InstanceOfName FB21200_POWDER_FLOW_SENSOR_MEDICOAT, InstanceOfType FB
"FB21200_POWDER_FLOW_SENSOR_MEDICOAT"
BEGIN
END_DATA_BLOCK

DATA_BLOCK "DB21209_UNIT_01_LASER_HEAD_MEDICOAT"   // DB21209
{ DB_Accessible_From_OPC_UA := 'FALSE' }
VERSION : 0.1
// stored: AutoNumber false, DBAccessibleFromOPCUA false, DBAccessibleFromWebserver true, InstanceOfName FB21200_POWDER_FLOW_SENSOR_MEDICOAT, InstanceOfType FB
"FB21200_POWDER_FLOW_SENSOR_MEDICOAT"
BEGIN
END_DATA_BLOCK

DATA_BLOCK "DB21210_UNIT_02_LASER_HEAD_MEDICOAT"   // DB21210
{ DB_Accessible_From_OPC_UA := 'FALSE' }
VERSION : 0.1
// stored: AutoNumber false, DBAccessibleFromOPCUA false, DBAccessibleFromWebserver true, InstanceOfName FB21200_POWDER_FLOW_SENSOR_MEDICOAT, InstanceOfType FB
"FB21200_POWDER_FLOW_SENSOR_MEDICOAT"
BEGIN
END_DATA_BLOCK

DATA_BLOCK "DB2002_BA_MODES_MG1"   // DB2002
{ DB_Accessible_From_OPC_UA := 'FALSE' }
VERSION : 0.1
// stored: AutoNumber false, DBAccessibleFromOPCUA false, DBAccessibleFromWebserver true, InstanceOfName FB2002_BA_MODE, InstanceOfType FB
"FB2002_BA_MODE"
BEGIN
END_DATA_BLOCK

DATA_BLOCK "DB2003_BA_MODES_MG2"   // DB2003
{ DB_Accessible_From_OPC_UA := 'FALSE' }
VERSION : 0.1
// stored: AutoNumber false, DBAccessibleFromOPCUA false, DBAccessibleFromWebserver true, InstanceOfName FB2002_BA_MODE, InstanceOfType FB
"FB2002_BA_MODE"
BEGIN
END_DATA_BLOCK
